	REGION B1.7.2
	    //B1.7.2
	    #"B1.7.2"(ConveyorID := _."B1.7.2",
	              ConveyorSensor:=_."ASiGW-MCC001-bw143-C1: Input"."Sensor B1.7.2",
	              Fault := DB_UDI.ProductionLine.Fault.Stop.Conveyor[_."B1.7.2"],
	              Upstream := DB_UDI.ProductionLine.Upstream.Conveyor[_."B1.7.2"],
	              Downstream := DB_UDI.ProductionLine.DownstreamAccu.Stop.Conveyor[_."B1.7.2"],
	              Interlock := DB_UDI.ProductionLine.Interlock.Stop.Conveyor[_."B1.7.2"],
	              RunForward=>_."ASiGW-MCC001-bw143-C1: Output"."Motor -B1.7.2",
	              WriteAsiDir=>_."ASiGW-MCC001-bw143-C1: Output"."Dir -B1.7.2");
	    
	END_REGION
	
	REGION B1.7.3
	    //B1.7.3
	    #"B1.7.3"(ConveyorID := _."B1.7.3",
	              ConveyorSensor:=_."ASiGW-MCC001-bw143-C1: Input"."Sensor B1.7.3",
	              Fault := DB_UDI.ProductionLine.Fault.Stop.Conveyor[_."B1.7.3"],
	              Upstream := DB_UDI.ProductionLine.Upstream.Conveyor[_."B1.7.3"],
	              Downstream := DB_UDI.ProductionLine.DownstreamAccu.Stop.Conveyor[_."B1.7.3"],
	              Interlock := DB_UDI.ProductionLine.Interlock.Stop.Conveyor[_."B1.7.3"],
	              RunForward=>_."ASiGW-MCC001-bw143-C1: Output"."Motor -B1.7.3",
	              WriteAsiDir=>_."ASiGW-MCC001-bw143-C1: Output"."Dir -B1.7.3");
	    
	END_REGION
	
	REGION B1.8.1
	    //B1.8.1
	    #"B1.8.1"(ConveyorID := _."B1.8.1",
	              ConveyorSensor:=_."ASiGW-MCC001-bw143-C2: Input"."Sensor B1.8.3",
	              Fault := DB_UDI.ProductionLine.Fault.Stop.Conveyor[_."B1.8.1"],
	              Upstream := DB_UDI.ProductionLine.Upstream.Conveyor[_."B1.8.1"],
	              Downstream := DB_UDI.ProductionLine.DownstreamAccu.Stop.Conveyor[_."B1.8.1"],
	              Interlock := DB_UDI.ProductionLine.Interlock.Stop.Conveyor[_."B1.8.1"],
	              RunForward => _."ASiGW-MCC001-bw143-C2: Output"."Motor B1.8.1",
	              WriteAsiDir => _."ASiGW-MCC001-bw143-C2: Output"."Dir B1.8.1");
	    
	END_REGION
	
	REGION B1.8.2
	    //B1.8.2
	    #"B1.8.2"(ConveyorID := _."B1.8.2",
	              ConveyorSensor:=_."ASiGW-MCC001-bw143-C2: Input"."Sensor B1.8.3",
	              Fault := DB_UDI.ProductionLine.Fault.Stop.Conveyor[_."B1.8.2"],
	              Upstream := DB_UDI.ProductionLine.Upstream.Conveyor[_."B1.8.2"],
	              Downstream := DB_UDI.ProductionLine.DownstreamAccu.Stop.Conveyor[_."B1.8.2"],
	              Interlock := DB_UDI.ProductionLine.Interlock.Stop.Conveyor[_."B1.8.2"],
	              RunForward=>_."ASiGW-MCC001-bw143-C2: Output"."Motor B1.8.2",
	              WriteAsiDir=>_."ASiGW-MCC001-bw143-C2: Output"."Dir B1.8.2");
	    
	END_REGION
	
	REGION B1.8.3
	    //B1.8.3
	    #"B1.8.3"(ConveyorID := _."B1.8.3",
	              ConveyorSensor:=_."ASiGW-MCC001-bw143-C2: Input"."Sensor B1.8.3",
	              Fault := DB_UDI.ProductionLine.Fault.Stop.Conveyor[_."B1.8.3"],
	              Upstream := DB_UDI.ProductionLine.Upstream.Conveyor[_."B1.8.3"],
	              Downstream := DB_UDI.ProductionLine.DownstreamAccu.Stop.Conveyor[_."B1.8.3"],
	              Interlock := DB_UDI.ProductionLine.Interlock.Stop.Conveyor[_."B1.8.3"],
	              RunForward=>_."ASiGW-MCC001-bw143-C2: Output"."Motor B1.8.3",
	              WriteAsiDir=>_."ASiGW-MCC001-bw143-C2: Output"."Dir B1.8.3");
	    
	END_REGION
	
	REGION B1.9.1
	    //// B1.9.1 (DP2)
	    #"B1.9.1"(ConveyorID := _."B1.9.1",
	              ConveyorSensor:=_."ASiGW-MCC001-bw143-C2: Input"."Sensor B1.9.1",
	              Fault := DB_UDI.ProductionLine.Fault.Stop.Conveyor[_."B1.9.1"],
	              Upstream := DB_UDI.ProductionLine.Upstream.Conveyor[_."B1.9.1"],
	              Downstream := DB_UDI.ProductionLine.DownstreamAccu.Stop.Conveyor[_."B1.9.1"],
	              Interlock := DB_UDI.ProductionLine.Interlock.Stop.Conveyor[_."B1.9.1"],
	              RunForward=>_."ASiGW-MCC001-bw143-C2: Output"."Motor B1.9.1",
	              WriteAsiDir=>_."ASiGW-MCC001-bw143-C2: Output"."Dir B1.9.1");
	    
	END_REGION
	
	REGION B1.9.2
	    //B1.9.2
	    #"B1.9.2"(ConveyorID := _."B1.9.2",
	              ConveyorSensor:=_."ASiGW-MCC001-bw143-C2: Input"."Sensor B1.9.2",
	              Fault := DB_UDI.ProductionLine.Fault.Stop.Conveyor[_."B1.9.2"],
	              Upstream := DB_UDI.ProductionLine.Upstream.Conveyor[_."B1.9.2"],
	              Downstream := DB_UDI.ProductionLine.DownstreamAccu.Stop.Conveyor[_."B1.9.2"],
	              Interlock := DB_UDI.ProductionLine.Interlock.Stop.Conveyor[_."B1.9.2"],
	              RunForward=>_."ASiGW-MCC001-bw143-C2: Output"."Motor B1.9.2",
	              WriteAsiDir=>_."ASiGW-MCC001-bw143-C2: Output"."Dir B1.9.2");
	    
	END_REGION
	
	REGION B1.10.1 Transfer Unit
	    //// Transfer B1.10.1
	    #"B1.10.1"(TransferID := _."B1.10.1",
	               TransferSensor:=_."ASiGW-MCC001-bw143-C2: Input"."LoadPresence -B1.10.1",
	               Fault := DB_UDI.ProductionLine.Fault.Stop.Conveyor[_."B1.10.1"],
	               Upstream := DB_UDI.ProductionLine.Upstream.Conveyor[_."B1.10.1"],
	               FrontSensor:=_."ASiGW-MCC001-bw143-C2: Input"."FrontSensor -B1.10.1",
	               EndSensor:=_."ASiGW-MCC001-bw143-C2: Input"."EndSensor -B1.10.1",
	               "Left/RightSensor":=_."ASiGW-MCC001-bw143-C2: Input"."LeftSensor -B1.10.1",
	               Downstream := DB_UDI.ProductionLine.DownstreamAccu.Stop.Conveyor[_."B1.10.1"],
	               TransferDirection := DB_ToteTracking.Conveyor[_."B1.10.1"].ToteDir,
	               StartSignal => _."ASiGW-MCC001-bw143-C2: Output"."StartSignal -B1.10.1",
	               Cmd1 => _."ASiGW-MCC001-bw143-C2: Output"."Command1 -B1.10.1",
	               Cmd2 => _."ASiGW-MCC001-bw143-C2: Output"."Command2 -B1.10.1",
	               ErrorReset => _."ASiGW-MCC001-bw143-C2: Output"."ErrorReset -B1.10.1");
	    
	END_REGION
	
	REGION B1.11.1
	    //// B1.11.1 (Go straight TR_B1.11.1)
	    #"B1.11.1"(ConveyorID := _."B1.11.1",
	               ConveyorSensor:=_."ASiGW-MCC001-bw143-C2: Input"."Sensor B1.11.1",
	               Fault := DB_UDI.ProductionLine.Fault.Stop.Conveyor[_."B1.11.1"],
	               Upstream := DB_UDI.ProductionLine.Upstream.Conveyor[_."B1.11.1"],
	               Downstream := DB_UDI.ProductionLine.DownstreamAccu.Stop.Conveyor[_."B1.11.1"],
	               Interlock := DB_UDI.ProductionLine.Interlock.Stop.Conveyor[_."B1.11.1"],
	               RunForward=>_."ASiGW-MCC001-bw143-C2: Output"."Motor B1.11.1",
	               WriteAsiDir=>_."ASiGW-MCC001-bw143-C2: Output"."Dir B1.11.1");
	    
	END_REGION
	
	REGION B1.11.2
	    //B1.11.2
	    #"B1.11.2"(ConveyorID := _."B1.11.2",
	               ConveyorSensor:=_."ASiGW-MCC001-bw143-C2: Input"."Sensor B1.11.4",
	               Fault := DB_UDI.ProductionLine.Fault.Stop.Conveyor[_."B1.11.2"],
	               Upstream := DB_UDI.ProductionLine.Upstream.Conveyor[_."B1.11.2"],
	               Downstream := DB_UDI.ProductionLine.DownstreamAccu.Stop.Conveyor[_."B1.11.2"],
	               Interlock := DB_UDI.ProductionLine.Interlock.Stop.Conveyor[_."B1.11.2"],
	               RunForward=>_."ASiGW-MCC001-bw143-C2: Output"."Motor B1.11.2",
	               WriteAsiDir=>_."ASiGW-MCC001-bw143-C2: Output"."Dir B1.11.2");
	    
	END_REGION
	
	REGION B1.11.3
	    //B1.11.3
	    #"B1.11.3"(ConveyorID := _."B1.11.3",
	               ConveyorSensor:=_."ASiGW-MCC001-bw143-C2: Input"."Sensor B1.11.4",
	               Fault := DB_UDI.ProductionLine.Fault.Stop.Conveyor[_."B1.11.3"],
	               Upstream := DB_UDI.ProductionLine.Upstream.Conveyor[_."B1.11.3"],
	               Downstream := DB_UDI.ProductionLine.DownstreamAccu.Stop.Conveyor[_."B1.11.3"],
	               Interlock := DB_UDI.ProductionLine.Interlock.Stop.Conveyor[_."B1.11.3"],
	               RunForward=>_."ASiGW-MCC001-bw143-C2: Output"."Motor B1.11.3",
	               WriteAsiDir=>_."ASiGW-MCC001-bw143-C2: Output"."Dir B1.11.3");
	    
	END_REGION
	
	REGION B1.11.4
	    //B1.11.4
	    #"B1.11.4"(ConveyorID := _."B1.11.4",
	               ConveyorSensor:=_."ASiGW-MCC001-bw143-C2: Input"."Sensor B1.11.4",
	               Fault := DB_UDI.ProductionLine.Fault.Stop.Conveyor[_."B1.11.4"],
	               Upstream := DB_UDI.ProductionLine.Upstream.Conveyor[_."B1.11.4"],
	               Downstream := DB_UDI.ProductionLine.DownstreamAccu.Stop.Conveyor[_."B1.11.4"],
	               Interlock := DB_UDI.ProductionLine.Interlock.Stop.Conveyor[_."B1.11.4"],
	               RunForward => _."ASiGW-MCC001-bw143-C2: Output"."Motor B1.11.4",
	               WriteAsiDir => _."ASiGW-MCC001-bw143-C2: Output"."Dir B1.11.4");
	    
	END_REGION
	
	REGION B1.12.1
	    //B1.12.1
	    #"B1.12.1"(ConveyorID := _."B1.12.1",
	               ConveyorSensor:=_."ASiGW-MCC001-bw143-C2: Input"."Sensor B1.12.1",
	               Fault := DB_UDI.ProductionLine.Fault.Stop.Conveyor[_."B1.12.1"],
	               Upstream := DB_UDI.ProductionLine.Upstream.Conveyor[_."B1.12.1"],
	               Downstream := DB_UDI.ProductionLine.DownstreamAccu.Stop.Conveyor[_."B1.12.1"],
	               Interlock := DB_UDI.ProductionLine.Interlock.Stop.Conveyor[_."B1.12.1"],
	               RunForward=>_."ASiGW-MCC001-bw143-C2: Output"."Motor B1.12.1",
	               WriteAsiDir=>_."ASiGW-MCC001-bw143-C2: Output"."Dir B1.12.1");
	    
	END_REGION
	
	REGION B1.12.2
	    //B1.12.2
	    #"B1.12.2"(ConveyorID := _."B1.12.2",
	               ConveyorSensor:=_."ASiGW-MCC001-bw143-C2: Input"."Sensor B1.12.2",
	               Fault := DB_UDI.ProductionLine.Fault.Stop.Conveyor[_."B1.12.2"],
	               Upstream := DB_UDI.ProductionLine.Upstream.Conveyor[_."B1.12.2"],
	               Downstream := DB_UDI.ProductionLine.DownstreamAccu.Stop.Conveyor[_."B1.12.2"],
	               Interlock := DB_UDI.ProductionLine.Interlock.Stop.Conveyor[_."B1.12.2"],
	               RunForward=>_."ASiGW-MCC001-bw143-C2: Output"."Motor B1.12.2",
	               WriteAsiDir=>_."ASiGW-MCC001-bw143-C2: Output"."Dir B1.12.2");
	    
	END_REGION
	
	REGION B1.13.1 Transfer Unit
	    //// Transfer B1.13.1
	    #"B1.13.1"(TransferID := _."B1.13.1",
	               TransferSensor:=_."ASiGW-MCC001-bw143-C2: Input"."LoadPresence -B1.13.1",
	               Fault := DB_UDI.ProductionLine.Fault.Stop.Conveyor[_."B1.13.1"],
	               Upstream := DB_UDI.ProductionLine.Upstream.Conveyor[_."B1.13.1"],
	               FrontSensor:=_."ASiGW-MCC001-bw143-C2: Input"."FrontSensor -B1.13.1",
	               EndSensor:=_."ASiGW-MCC001-bw143-C2: Input"."EndSensor -B1.13.1",
	               "Left/RightSensor":=_."ASiGW-MCC001-bw143-C2: Input"."LeftSensor -B1.13.1",
	               Downstream := DB_UDI.ProductionLine.DownstreamAccu.Stop.Conveyor[_."B1.13.1"],
	               TransferDirection := DB_ToteTracking.Conveyor[_."B1.13.1"].ToteDir,
	               StartSignal => _."ASiGW-MCC001-bw143-C2: Output"."StartSignal - B1.13.1",
	               Cmd1 => _."ASiGW-MCC001-bw143-C2: Output"."Command1 -B1.13.1",
	               Cmd2 => _."ASiGW-MCC001-bw143-C2: Output"."Command2 -B1.13.1",
	               ErrorReset => _."ASiGW-MCC001-bw143-C2: Output"."ErrorReset -B1.13.1");
	    
	END_REGION
	
	REGION B1.14.1 Transfer Unit
	    //// Transfer B1.14.1
	    #"B1.14.1"(TransferID := _."B1.14.1",
	               TransferSensor:=_."ASiGW-MCC001-bw143-C2: Input"."LoadPresence -B1.14.1",
	               Fault := DB_UDI.ProductionLine.Fault.Stop.Conveyor[_."B1.14.1"],
	               Upstream := DB_UDI.ProductionLine.Upstream.Conveyor[_."B1.14.1"],
	               FrontSensor:=_."ASiGW-MCC001-bw143-C2: Input"."FrontSensor -B1.14.1",
	               EndSensor:=_."ASiGW-MCC001-bw143-C2: Input"."EndSensor -B1.14.1",
	               "Left/RightSensor":=_."ASiGW-MCC001-bw143-C2: Input"."LeftSensor -B1.14.1",
	               Downstream := DB_UDI.ProductionLine.DownstreamAccu.Stop.Conveyor[_."B1.14.1"],
	               TransferDirection := DB_ToteTracking.Conveyor[_."B1.14.1"].ToteDir,
	               StartSignal => _."ASiGW-MCC001-bw143-C2: Output"."StartSignal -B1.14.1",
	               Cmd1 => _."ASiGW-MCC001-bw143-C2: Output"."Command1 -B1.14.1",
	               Cmd2 => _."ASiGW-MCC001-bw143-C2: Output"."Command2 -B1.14.1",
	               ErrorReset => _."ASiGW-MCC001-bw143-C2: Output"."ErrorReset -B1.14.1");
	    
	END_REGION
	
	REGION B1.15.1
	    //// B1.15.1 (Go straight TR_B1.17.1)
	    #"B1.15.1"(ConveyorID := _."B1.15.1",
	               ConveyorSensor:=_."ASiGW-MCC001-bw143-C2: Input"."Sensor B1.15.1",
	               Fault := DB_UDI.ProductionLine.Fault.Stop.Conveyor[_."B1.15.1"],
	               Upstream := DB_UDI.ProductionLine.Upstream.Conveyor[_."B1.15.1"],
	               Downstream := DB_UDI.ProductionLine.DownstreamAccu.Stop.Conveyor[_."B1.15.1"],
	               Interlock := DB_UDI.ProductionLine.Interlock.Stop.Conveyor[_."B1.15.1"],
	               RunForward=>_."ASiGW-MCC001-bw143-C2: Output"."Motor B1.15.1",
	               WriteAsiDir=>_."ASiGW-MCC001-bw143-C2: Output"."Dir B1.15.1");
	    
	END_REGION
	
	REGION B1.15.2
	    //B1.15.2
	    #"B1.15.2"(ConveyorID := _."B1.15.2",
	               ConveyorSensor:=_."ASiGW-MCC001-bw143-C2: Input"."Sensor B1.15.2",
	               Fault := DB_UDI.ProductionLine.Fault.Stop.Conveyor[_."B1.15.2"],
	               Upstream := DB_UDI.ProductionLine.Upstream.Conveyor[_."B1.15.2"],
	               Downstream := DB_UDI.ProductionLine.DownstreamAccu.Stop.Conveyor[_."B1.15.2"],
	               Interlock := DB_UDI.ProductionLine.Interlock.Stop.Conveyor[_."B1.15.2"],
	               RunForward=>_."ASiGW-MCC001-bw143-C2: Output"."Motor B1.15.2",
	               WriteAsiDir=>_."ASiGW-MCC001-bw143-C2: Output"."Dir B1.15.2");
	    
	END_REGION
	
	REGION B1.16.1
	    //B1.16.1
	    #"B1.16.1"(ConveyorID := _."B1.16.1",
	               ConveyorSensor:=_."ASiGW-MCC001-bw143-C2: Input"."Sensor B1.16.8",
	               Fault := DB_UDI.ProductionLine.Fault.Stop.Conveyor[_."B1.16.1"],
	               Upstream := DB_UDI.ProductionLine.Upstream.Conveyor[_."B1.16.1"],
	               Downstream := DB_UDI.ProductionLine.DownstreamAccu.Stop.Conveyor[_."B1.16.1"],
	               Interlock := DB_UDI.ProductionLine.Interlock.Stop.Conveyor[_."B1.16.1"],
	               RunForward => _."ASiGW-MCC001-bw143-C2: Output"."Motor B1.16.1",
	               WriteAsiDir => _."ASiGW-MCC001-bw143-C2: Output"."Dir B1.16.1");
	    
	END_REGION
	
	REGION B1.16.2
	    //B1.16.2
	    #"B1.16.2"(ConveyorID := _."B1.16.2",
	               ConveyorSensor:=_."ASiGW-MCC001-bw143-C2: Input"."Sensor B1.16.8",
	               Fault := DB_UDI.ProductionLine.Fault.Stop.Conveyor[_."B1.16.2"],
	               Upstream := DB_UDI.ProductionLine.Upstream.Conveyor[_."B1.16.2"],
	               Downstream := DB_UDI.ProductionLine.DownstreamAccu.Stop.Conveyor[_."B1.16.2"],
	               Interlock := DB_UDI.ProductionLine.Interlock.Stop.Conveyor[_."B1.16.2"],
	               RunForward=>_."ASiGW-MCC001-bw143-C2: Output"."Motor B1.16.2",
	               WriteAsiDir=>_."ASiGW-MCC001-bw143-C2: Output"."Dir B1.16.2");
	    
	END_REGION
	
	REGION B1.16.3
	    //B1.16.3
	    #"B1.16.3"(ConveyorID := _."B1.16.3",
	               ConveyorSensor:=_."ASiGW-MCC001-bw143-C2: Input"."Sensor B1.16.8",
	               Fault := DB_UDI.ProductionLine.Fault.Stop.Conveyor[_."B1.16.3"],
	               Upstream := DB_UDI.ProductionLine.Upstream.Conveyor[_."B1.16.3"],
	               Downstream := DB_UDI.ProductionLine.DownstreamAccu.Stop.Conveyor[_."B1.16.3"],
	               Interlock := DB_UDI.ProductionLine.Interlock.Stop.Conveyor[_."B1.16.3"],
	               RunForward=>_."ASiGW-MCC001-bw143-C2: Output"."Motor B1.16.3",
	               WriteAsiDir=>_."ASiGW-MCC001-bw143-C2: Output"."Dir B1.16.3");
	    
	END_REGION
	
	REGION B1.16.4
	    //B1.16.4
	    #"B1.16.4"(ConveyorID := _."B1.16.4",
	               ConveyorSensor:=_."ASiGW-MCC001-bw143-C2: Input"."Sensor B1.16.8",
	               Fault := DB_UDI.ProductionLine.Fault.Stop.Conveyor[_."B1.16.4"],
	               Upstream := DB_UDI.ProductionLine.Upstream.Conveyor[_."B1.16.4"],
	               Downstream := DB_UDI.ProductionLine.DownstreamAccu.Stop.Conveyor[_."B1.16.4"],
	               Interlock := DB_UDI.ProductionLine.Interlock.Stop.Conveyor[_."B1.16.4"],
	               RunForward=>_."ASiGW-MCC001-bw143-C2: Output"."Motor B1.16.4",
	               WriteAsiDir=>_."ASiGW-MCC001-bw143-C2: Output"."Dir B1.16.4");
	    
	END_REGION
	
	REGION B1.16.5
	    //B1.16.5
	    #"B1.16.5"(ConveyorID := _."B1.16.5",
	               ConveyorSensor:=_."ASiGW-MCC001-bw143-C2: Input"."Sensor B1.16.8",
	               Fault := DB_UDI.ProductionLine.Fault.Stop.Conveyor[_."B1.16.5"],
	               Upstream := DB_UDI.ProductionLine.Upstream.Conveyor[_."B1.16.5"],
	               Downstream := DB_UDI.ProductionLine.DownstreamAccu.Stop.Conveyor[_."B1.16.5"],
	               Interlock := DB_UDI.ProductionLine.Interlock.Stop.Conveyor[_."B1.16.5"],
	               RunForward=>_."ASiGW-MCC001-bw143-C2: Output"."Motor B1.16.5",
	               WriteAsiDir=>_."ASiGW-MCC001-bw143-C2: Output"."Dir B1.16.5");
	    
	END_REGION
	
	REGION B1.16.6
	    //B1.16.6
	    #"B1.16.6"(ConveyorID := _."B1.16.6",
	               ConveyorSensor:=_."ASiGW-MCC001-bw143-C2: Input"."Sensor B1.16.8",
	               Fault := DB_UDI.ProductionLine.Fault.Stop.Conveyor[_."B1.16.6"],
	               Upstream := DB_UDI.ProductionLine.Upstream.Conveyor[_."B1.16.6"],
	               Downstream := DB_UDI.ProductionLine.DownstreamAccu.Stop.Conveyor[_."B1.16.6"],
	               Interlock := DB_UDI.ProductionLine.Interlock.Stop.Conveyor[_."B1.16.6"],
	               RunForward=>_."ASiGW-MCC001-bw143-C2: Output"."Motor B1.16.6",
	               WriteAsiDir=>_."ASiGW-MCC001-bw143-C2: Output"."Dir B1.16.6");
	    
	END_REGION
	
	REGION B1.16.7
	    //B1.16.7
	    #"B1.16.7"(ConveyorID := _."B1.16.7",
	               ConveyorSensor:=_."ASiGW-MCC001-bw143-C2: Input"."Sensor B1.16.8",
	               Fault := DB_UDI.ProductionLine.Fault.Stop.Conveyor[_."B1.16.7"],
	               Upstream := DB_UDI.ProductionLine.Upstream.Conveyor[_."B1.16.7"],
	               Downstream := DB_UDI.ProductionLine.DownstreamAccu.Stop.Conveyor[_."B1.16.7"],
	               Interlock := DB_UDI.ProductionLine.Interlock.Stop.Conveyor[_."B1.16.7"],
	               RunForward => _."ASiGW-MCC001-bw143-C2: Output"."Motor B1.16.7",
	               WriteAsiDir => _."ASiGW-MCC001-bw143-C2: Output"."Dir B1.16.7");
	    
	END_REGION
	
	REGION B1.16.8
	    //B1.16.8
	    #"B1.16.8"(ConveyorID := _."B1.16.8",
	               ConveyorSensor:=_."ASiGW-MCC001-bw143-C2: Input"."Sensor B1.16.8",
	               Fault := DB_UDI.ProductionLine.Fault.Stop.Conveyor[_."B1.16.8"],
	               Upstream := DB_UDI.ProductionLine.Upstream.Conveyor[_."B1.16.8"],
	               Downstream := DB_UDI.ProductionLine.DownstreamAccu.Stop.Conveyor[_."B1.16.8"],
	               Interlock := DB_UDI.ProductionLine.Interlock.Stop.Conveyor[_."B1.16.8"],
	               RunForward=>_."ASiGW-MCC001-bw143-C2: Output"."Motor B1.16.8",
	               WriteAsiDir=>_."ASiGW-MCC001-bw143-C2: Output"."Dir B1.16.8");
	    
	END_REGION
	
	REGION B1.17.1
	    //// B1.17.1 (DP3)
	    #"B1.17.1"(ConveyorID := _."B1.17.1",
	               ConveyorSensor:=_."ASiGW-MCC001-bw143-C2: Input"."Sensor B1.17.1",
	               Fault := DB_UDI.ProductionLine.Fault.Stop.Conveyor[_."B1.17.1"],
	               Upstream := DB_UDI.ProductionLine.Upstream.Conveyor[_."B1.17.1"],
	               Downstream := DB_UDI.ProductionLine.DownstreamAccu.Stop.Conveyor[_."B1.17.1"],
	               Interlock := DB_UDI.ProductionLine.Interlock.Stop.Conveyor[_."B1.17.1"],
	               RunForward => _."ASiGW-MCC001-bw143-C2: Output"."Motor B1.17.1",
	               WriteAsiDir => _."ASiGW-MCC001-bw143-C2: Output"."Dir B1.17.1");
	    
	END_REGION
	
	REGION B1.17.2
	    //B1.17.2
	    #"B1.17.2"(ConveyorID := _."B1.17.2",
	               ConveyorSensor:=_."ASiGW-MCC001-bw143-C2: Input"."Sensor B1.17.2",
	               Fault := DB_UDI.ProductionLine.Fault.Stop.Conveyor[_."B1.17.2"],
	               Upstream := DB_UDI.ProductionLine.Upstream.Conveyor[_."B1.17.2"],
	               Downstream := DB_UDI.ProductionLine.DownstreamAccu.Stop.Conveyor[_."B1.17.2"],
	               Interlock := DB_UDI.ProductionLine.Interlock.Stop.Conveyor[_."B1.17.2"],
	               RunForward => _."ASiGW-MCC001-bw143-C2: Output"."Motor B1.17.2",
	               WriteAsiDir => _."ASiGW-MCC001-bw143-C2: Output"."Dir B1.17.2");
	    
	END_REGION
	
	REGION B1.17.3
	    //B1.17.3
	    #"B1.17.3"(ConveyorID := _."B1.17.3",
	               ConveyorSensor:=_."ASiGW-MCC001-bw143-C2: Input"."Sensor B1.17.3",
	               Fault := DB_UDI.ProductionLine.Fault.Stop.Conveyor[_."B1.17.3"],
	               Upstream := DB_UDI.ProductionLine.Upstream.Conveyor[_."B1.17.3"],
	               Downstream := DB_UDI.ProductionLine.DownstreamAccu.Stop.Conveyor[_."B1.17.3"],
	               Interlock := DB_UDI.ProductionLine.Interlock.Stop.Conveyor[_."B1.17.3"],
	               RunForward => _."ASiGW-MCC001-bw143-C2: Output"."Motor B1.17.3",
	               WriteAsiDir => _."ASiGW-MCC001-bw143-C2: Output"."Dir B1.17.3");
	    
	END_REGION
	
	REGION B1.17.4
	    //B1.17.4
	    #"B1.17.4"(ConveyorID := _."B1.17.4",
	               ConveyorSensor:=_."ASiGW-MCC001-bw143-C2: Input"."Sensor B1.17.4",
	               Fault := DB_UDI.ProductionLine.Fault.Stop.Conveyor[_."B1.17.4"],
	               Upstream := DB_UDI.ProductionLine.Upstream.Conveyor[_."B1.17.4"],
	               Downstream := DB_UDI.ProductionLine.DownstreamAccu.Stop.Conveyor[_."B1.17.4"],
	               Interlock := DB_UDI.ProductionLine.Interlock.Stop.Conveyor[_."B1.17.4"],
	               RunForward => _."ASiGW-MCC001-bw143-C2: Output"."Motor B1.17.4",
	               WriteAsiDir => _."ASiGW-MCC001-bw143-C2: Output"."Dir B1.17.4");
	    
	END_REGION
	
	REGION B1.18.1 Transfer Unit
	    //// Transfer B1.18.1
	    #"B1.18.1"(TransferID := _."B1.18.1",
	               TransferSensor:=_."ASiGW-MCC001-bw143-C2: Input"."LoadPresence -B1.18.1",
	               Fault := DB_UDI.ProductionLine.Fault.Stop.Conveyor[_."B1.18.1"],
	               Upstream := DB_UDI.ProductionLine.Upstream.Conveyor[_."B1.18.1"],
	               FrontSensor:=_."ASiGW-MCC001-bw143-C2: Input"."FrontSensor -B1.18.1",
	               EndSensor:=_."ASiGW-MCC001-bw143-C2: Input"."EndSensor -B1.18.1",
	               "Left/RightSensor":=_."ASiGW-MCC001-bw143-C2: Input"."LeftSensor -B1.18.1",
	               Downstream := DB_UDI.ProductionLine.DownstreamAccu.Stop.Conveyor[_."B1.18.1"],
	               TransferDirection := DB_ToteTracking.Conveyor[_."B1.18.1"].ToteDir,
	               StartSignal => _."ASiGW-MCC001-bw143-C2: Output"."StartSignal -B1.18.1",
	               Cmd1 => _."ASiGW-MCC001-bw143-C2: Output"."Command1 -B1.18.1",
	               Cmd2 => _."ASiGW-MCC001-bw143-C2: Output"."Command2 -B1.18.1",
	               ErrorReset => _."ASiGW-MCC001-bw143-C2: Output"."ErrorReset -B1.18.1");
	    
	END_REGION
	
	REGION B1.19.1
	    //B1.19.1
	    #"B1.19.1"(ConveyorID := _."B1.19.1",
	               ConveyorSensor:=_."ASiGW-MCC001-bw143-C2: Input"."Sensor B1.19.1",
	               Fault := DB_UDI.ProductionLine.Fault.Stop.Conveyor[_."B1.19.1"],
	               Upstream := DB_UDI.ProductionLine.Upstream.Conveyor[_."B1.19.1"],
	               Downstream := DB_UDI.ProductionLine.DownstreamAccu.Stop.Conveyor[_."B1.19.1"],
	               Interlock := DB_UDI.ProductionLine.Interlock.Stop.Conveyor[_."B1.19.1"],
	               RunForward => _."ASiGW-MCC001-bw143-C2: Output"."Motor B1.19.1",
	               WriteAsiDir => _."ASiGW-MCC001-bw143-C2: Output"."Dir B1.19.1");
	    
	END_REGION
	
	REGION B1.20.1
	    //B1.20.1
	    #"B1.20.1"(ConveyorID := _."B1.20.1",
	               ConveyorSensor:=_."ASiGW-MCC001-bw143-C2: Input"."Sensor B1.20.1",
	               Fault := DB_UDI.ProductionLine.Fault.Stop.Conveyor[_."B1.20.1"],
	               Upstream := DB_UDI.ProductionLine.Upstream.Conveyor[_."B1.20.1"],
	               Downstream := DB_UDI.ProductionLine.DownstreamAccu.Stop.Conveyor[_."B1.20.1"],
	               Interlock := DB_UDI.ProductionLine.Interlock.Stop.Conveyor[_."B1.20.1"],
	               RunForward => _."ASiGW-MCC001-bw143-C2: Output"."Motor B1.20.1",
	               WriteAsiDir => _."ASiGW-MCC001-bw143-C2: Output"."Dir B1.20.1");
	    
	END_REGION
	
	REGION B1.20.2
	    //B1.20.2
	    #"B1.20.2"(ConveyorID := _."B1.20.2",
	               ConveyorSensor:=_."ASiGW-MCC001-bw143-C2: Input"."Sensor B1.20.2",
	               Fault := DB_UDI.ProductionLine.Fault.Stop.Conveyor[_."B1.20.2"],
	               Upstream := DB_UDI.ProductionLine.Upstream.Conveyor[_."B1.20.2"],
	               Downstream := DB_UDI.ProductionLine.DownstreamAccu.Stop.Conveyor[_."B1.20.2"],
	               Interlock := DB_UDI.ProductionLine.Interlock.Stop.Conveyor[_."B1.20.2"],
	               RunForward => _."ASiGW-MCC001-bw143-C2: Output"."Motor B1.20.2",
	               WriteAsiDir => _."ASiGW-MCC001-bw143-C2: Output"."Dir B1.20.2");
	    
	END_REGION
	
	REGION B1.21.1
	    //B1.21.1
	    #"B1.21.1"(ConveyorID := _."B1.21.1",
	               ConveyorSensor:=_."ASiGW-MCC001-bw143-C2: Input"."Sensor B1.21.1",
	               Fault := DB_UDI.ProductionLine.Fault.Stop.Conveyor[_."B1.21.1"],
	               Upstream := DB_UDI.ProductionLine.Upstream.Conveyor[_."B1.21.1"],
	               Downstream := DB_UDI.ProductionLine.DownstreamAccu.Stop.Conveyor[_."B1.21.1"],
	               Interlock := DB_UDI.ProductionLine.Interlock.Stop.Conveyor[_."B1.21.1"],
	               RunForward => _."ASiGW-MCC001-bw143-C2: Output"."Motor B1.21.1",
	               WriteAsiDir => _."ASiGW-MCC001-bw143-C2: Output"."Dir B1.21.1");
	    
	END_REGION
	
	REGION B1.21.2
	    //B1.21.2
	    #"B1.21.2"(ConveyorID := _."B1.21.2",
	               ConveyorSensor:=_."ASiGW-MCC001-bw143-C2: Input"."Sensor B1.21.2",
	               Fault := DB_UDI.ProductionLine.Fault.Stop.Conveyor[_."B1.21.2"],
	               Upstream := DB_UDI.ProductionLine.Upstream.Conveyor[_."B1.21.2"],
	               Downstream := DB_UDI.ProductionLine.DownstreamAccu.Stop.Conveyor[_."B1.21.2"],
	               Interlock := DB_UDI.ProductionLine.Interlock.Stop.Conveyor[_."B1.21.2"],
	               RunForward => _."ASiGW-MCC001-bw143-C2: Output"."Motor B1.21.2",
	               WriteAsiDir => _."ASiGW-MCC001-bw143-C2: Output"."Dir B1.21.2");
	    
	END_REGION
	
	REGION B1.21.3
	    //B1.21.3
	    #"B1.21.3"(ConveyorID := _."B1.21.3",
	               ConveyorSensor:=_."ASiGW-MCC001-bw143-C2: Input"."Sensor B1.23.1",
	               Fault := DB_UDI.ProductionLine.Fault.Stop.Conveyor[_."B1.21.3"],
	               Upstream := DB_UDI.ProductionLine.Upstream.Conveyor[_."B1.21.3"],
	               Downstream := DB_UDI.ProductionLine.DownstreamAccu.Stop.Conveyor[_."B1.21.3"],
	               Interlock := DB_UDI.ProductionLine.Interlock.Stop.Conveyor[_."B1.21.3"],
	               RunForward => _."ASiGW-MCC001-bw143-C2: Output"."Motor B1.21.3",
	               WriteAsiDir => _."ASiGW-MCC001-bw143-C2: Output"."Dir B1.21.3");
	    
	END_REGION
	
	REGION B1.22.1
	    //B1.22.1
	    #"B1.22.1"(ConveyorID := _."B1.22.1",
	               ConveyorSensor:=_."ASiGW-MCC001-bw143-C2: Input"."Sensor B1.23.1",
	               Fault := DB_UDI.ProductionLine.Fault.Stop.Conveyor[_."B1.22.1"],
	               Upstream := DB_UDI.ProductionLine.Upstream.Conveyor[_."B1.22.1"],
	               Downstream := DB_UDI.ProductionLine.DownstreamAccu.Stop.Conveyor[_."B1.22.1"],
	               Interlock := DB_UDI.ProductionLine.Interlock.Stop.Conveyor[_."B1.22.1"],
	               RunForward => _."ASiGW-MCC001-bw143-C2: Output"."Motor - B1.22.1",
	               WriteAsiDir => _."ASiGW-MCC001-bw143-C2: Output"."2-30A Dir",
	               WriteAsiSpeed => _."ASiGW-MCC001-bw143-C2: Output"."2-30A Speed");
	    
	END_REGION
	
	REGION B1.23.1
	    ////B1.23.1 Arm for Merger1
	    #"B1.23.1"(ConveyorID := _."B1.23.1",
	               ConveyorSensor:=_."ASiGW-MCC001-bw143-C2: Input"."Sensor B1.23.1",
	               Fault := DB_UDI.ProductionLine.Fault.Stop.Conveyor[_."B1.23.1"],
	               Upstream := DB_UDI.ProductionLine.Upstream.Conveyor[_."B1.23.1"],
	               Downstream := DB_UDI.ProductionLine.DownstreamAccu.Stop.Conveyor[_."B1.23.1"],
	               Interlock := DB_UDI.ProductionLine.Interlock.Stop.Conveyor[_."B1.23.1"],
	               RunForward => _."ASiGW-MCC001-bw143-C2: Output"."Motor B1.23.1",
	               WriteAsiDir => _."ASiGW-MCC001-bw143-C2: Output"."Dir B1.23.1");
	    
	END_REGION
	
	REGION C1.3.1 Transfer Unit
	    ////Transfer C1.3.1
	    #"C1.3.1"(TransferID := _."C1.3.1",
	              TransferSensor:=_."ASiGW-MCC001-bw143-C2: Input"."LoadPresence -C1.3.1",
	              Fault := DB_UDI.ProductionLine.Fault.Stop.Conveyor[_."C1.3.1"],
	              Upstream := DB_UDI.ProductionLine.Upstream.Conveyor[_."C1.3.1"],
	              FrontSensor:=_."ASiGW-MCC001-bw143-C2: Input"."FrontSensor -C1.3.1",
	              EndSensor:=_."ASiGW-MCC001-bw143-C2: Input"."EndSensor -C1.3.1",
	              "Left/RightSensor":=_."ASiGW-MCC001-bw143-C2: Input"."LeftSensor -C1.3.1",
	              Downstream := DB_UDI.ProductionLine.DownstreamAccu.Stop.Conveyor[_."C1.3.1"],
	              TransferDirection := DB_ToteTracking.Conveyor[_."C1.3.1"].ToteDir,
	              StartSignal => _."ASiGW-MCC001-bw143-C2: Output"."StartSignal -C1.3.1",
	              Cmd1 => _."ASiGW-MCC001-bw143-C2: Output"."Command1 -C1.3.1",
	              Cmd2 => _."ASiGW-MCC001-bw143-C2: Output"."Command2 -C1.3.1",
	              ErrorReset => _."ASiGW-MCC001-bw143-C2: Output"."ErrorReset -C1.3.1");
	    
	END_REGION
	
	REGION C1.2.2
	    //// C1.2.2  (Go Right TR_C1.1.3)
	    #"C1.2.2"(ConveyorID := _."C1.2.2",
	              ConveyorSensor:=_."ASiGW-MCC001-bw143-C2: Input"."Sensor C1.2.2",
	              Fault := DB_UDI.ProductionLine.Fault.Stop.Conveyor[_."C1.2.2"],
	              Upstream := DB_UDI.ProductionLine.Upstream.Conveyor[_."C1.2.2"],
	              Downstream := DB_UDI.ProductionLine.DownstreamAccu.Stop.Conveyor[_."C1.2.2"],
	              Interlock := DB_UDI.ProductionLine.Interlock.Stop.Conveyor[_."C1.2.2"],
	              RunForward=>_."ASiGW-MCC001-bw143-C2: Output"."Motor C1.2.2",
	              WriteAsiDir=>_."ASiGW-MCC001-bw143-C2: Output"."Dir C1.2.2");
	    
	END_REGION
	
	REGION C1.2.1
	    //C1.2.1
	    #"C1.2.1"(ConveyorID := _."C1.2.1",
	              ConveyorSensor:=_."ASiGW-MCC001-bw143-C2: Input"."Sensor C1.2.1",
	              Fault := DB_UDI.ProductionLine.Fault.Stop.Conveyor[_."C1.2.1"],
	              Upstream := DB_UDI.ProductionLine.Upstream.Conveyor[_."C1.2.1"],
	              Downstream := DB_UDI.ProductionLine.DownstreamAccu.Stop.Conveyor[_."C1.2.1"],
	              Interlock := DB_UDI.ProductionLine.Interlock.Stop.Conveyor[_."C1.2.1"],
	              RunForward=>_."ASiGW-MCC001-bw143-C2: Output"."Motor C1.2.1",
	              WriteAsiDir=>_."ASiGW-MCC001-bw143-C2: Output"."Dir C1.2.1");
	    
	END_REGION
	
	REGION C1.4.1
	    //// C1.4.1  (Go Left TR_C1.1.3)
	    #"C1.4.1"(ConveyorID := _."C1.4.1",
	              ConveyorSensor:=_."ASiGW-MCC001-bw143-C2: Input"."Sensor C1.4.1",
	              Fault := DB_UDI.ProductionLine.Fault.Stop.Conveyor[_."C1.4.1"],
	              Upstream := DB_UDI.ProductionLine.Upstream.Conveyor[_."C1.4.1"],
	              Downstream := DB_UDI.ProductionLine.DownstreamAccu.Stop.Conveyor[_."C1.4.1"],
	              Interlock := DB_UDI.ProductionLine.Interlock.Stop.Conveyor[_."C1.4.1"],
	              RunForward=>_."ASiGW-MCC001-bw143-C2: Output"."Motor C1.4.1",
	              WriteAsiDir=>_."ASiGW-MCC001-bw143-C2: Output"."Dir C1.4.1");
	    
	END_REGION
	
	REGION C1.4.2
	    //C1.4.2
	    #"C1.4.2"(ConveyorID := _."C1.4.2",
	              ConveyorSensor:=_."ASiGW-MCC001-bw143-C2: Input"."Sensor C1.4.2",
	              Fault := DB_UDI.ProductionLine.Fault.Stop.Conveyor[_."C1.4.2"],
	              Upstream := DB_UDI.ProductionLine.Upstream.Conveyor[_."C1.4.2"],
	              Downstream := DB_UDI.ProductionLine.DownstreamAccu.Stop.Conveyor[_."C1.4.2"],
	              Interlock := DB_UDI.ProductionLine.Interlock.Stop.Conveyor[_."C1.4.2"],
	              RunForward=>_."ASiGW-MCC001-bw143-C2: Output"."Motor C1.4.2",
	              WriteAsiDir=>_."ASiGW-MCC001-bw143-C2: Output"."Dir C1.4.2");
	    
	END_REGION
	
	REGION D1.1.1
	    ////  D1.1.1 (Go Right DP4)
	    #"D1.1.1"(ConveyorID := _."D1.1.1",
	              ConveyorSensor:=_."ASiGW-MCC001-bw200-C1: Input"."Sensor D1.2.1",
	              Fault := DB_UDI.ProductionLine.Fault.Stop.Conveyor[_."D1.1.1"],
	              Upstream := DB_UDI.ProductionLine.Upstream.Conveyor[_."D1.1.1"],
	              Downstream := DB_UDI.ProductionLine.DownstreamAccu.Stop.Conveyor[_."D1.1.1"],
	              Interlock := DB_UDI.ProductionLine.Interlock.Stop.Conveyor[_."D1.1.1"],
	              RunForward=>_."ASiGW-MCC001-bw200-C1: Output"."Motor D1.1.1",
	              WriteAsiDir=>_."ASiGW-MCC001-bw200-C1: Output"."Dir D1.1.1");
	    
	END_REGION
	
	REGION D1.2.1
	    //D1.2.1
	    #"D1.2.1"(ConveyorID := _."D1.2.1",
	              ConveyorSensor:=_."ASiGW-MCC001-bw200-C1: Input"."Sensor D1.2.1",
	              Fault := DB_UDI.ProductionLine.Fault.Stop.Conveyor[_."D1.2.1"],
	              Upstream := DB_UDI.ProductionLine.Upstream.Conveyor[_."D1.2.1"],
	              Downstream := DB_UDI.ProductionLine.DownstreamAccu.Stop.Conveyor[_."D1.2.1"],
	              Interlock := DB_UDI.ProductionLine.Interlock.Stop.Conveyor[_."D1.2.1"],
	              RunForward=>_."ASiGW-MCC001-bw200-C1: Output"."Motor - D1.2.1",
	              WriteAsiDir=>_."ASiGW-MCC001-bw200-C1: Output"."1-2A Dir",
	              WriteAsiSpeed=>_."ASiGW-MCC001-bw200-C1: Output"."1-2A Speed");
	    
	END_REGION
	
	REGION D1.3.1
	    //D1.3.1
	    #"D1.3.1"(ConveyorID := _."D1.3.1",
	              ConveyorSensor:=_."ASiGW-MCC001-bw200-C1: Input"."Sensor D1.3.1",
	              Fault := DB_UDI.ProductionLine.Fault.Stop.Conveyor[_."D1.3.1"],
	              Upstream := DB_UDI.ProductionLine.Upstream.Conveyor[_."D1.3.1"],
	              Downstream := DB_UDI.ProductionLine.DownstreamAccu.Stop.Conveyor[_."D1.3.1"],
	              Interlock := DB_UDI.ProductionLine.Interlock.Stop.Conveyor[_."D1.3.1"],
	              RunForward=>_."ASiGW-MCC001-bw200-C1: Output"."Motor - D1.3.1",
	              WriteAsiDir=>_."ASiGW-MCC001-bw200-C1: Output"."1-2A Dir",
	              WriteAsiSpeed=>_."ASiGW-MCC001-bw200-C1: Output"."1-2A Speed");
	    
	END_REGION
	
	REGION D1.4.1
	    //D1.4.1
	    #"D1.4.1"(ConveyorID := _."D1.4.1",
	              ConveyorSensor:=_."ASiGW-MCC001-bw200-C1: Input"."Sensor D1.4.1",
	              Fault := DB_UDI.ProductionLine.Fault.Stop.Conveyor[_."D1.4.1"],
	              Upstream := DB_UDI.ProductionLine.Upstream.Conveyor[_."D1.4.1"],
	              Downstream := DB_UDI.ProductionLine.DownstreamAccu.Stop.Conveyor[_."D1.4.1"],
	              Interlock := DB_UDI.ProductionLine.Interlock.Stop.Conveyor[_."D1.4.1"],
	              RunForward=>_."ASiGW-MCC001-bw200-C1: Output"."Motor D1.4.1",
	              WriteAsiDir=>_."ASiGW-MCC001-bw200-C1: Output"."Dir D1.4.1");
	    
	END_REGION
	
	REGION D1.5.1
	    //D1.5.1
	    #"D1.5.1"(ConveyorID := _."D1.5.1",
	              ConveyorSensor:=_."ASiGW-MCC001-bw200-C1: Input"."Sensor D1.5.1",
	              Fault := DB_UDI.ProductionLine.Fault.Stop.Conveyor[_."D1.5.1"],
	              Upstream := DB_UDI.ProductionLine.Upstream.Conveyor[_."D1.5.1"],
	              Downstream := DB_UDI.ProductionLine.DownstreamAccu.Stop.Conveyor[_."D1.5.1"],
	              Interlock := DB_UDI.ProductionLine.Interlock.Stop.Conveyor[_."D1.5.1"],
	              RunForward=>_."ASiGW-MCC001-bw200-C1: Output"."Motor - D1.5.1",
	              WriteAsiDir=>_."ASiGW-MCC001-bw200-C1: Output"."1-4A Dir",
	              WriteAsiSpeed=>_."ASiGW-MCC001-bw200-C1: Output"."1-4A Speed");
	    
	END_REGION
	
	REGION D1.6.1
	    //D1.6.1
	    #"D1.6.1"(ConveyorID := _."D1.6.1",
	              ConveyorSensor:=_."ASiGW-MCC001-bw200-C1: Input"."Sensor D1.6.1",
	              Fault := DB_UDI.ProductionLine.Fault.Stop.Conveyor[_."D1.6.1"],
	              Upstream := DB_UDI.ProductionLine.Upstream.Conveyor[_."D1.6.1"],
	              Downstream := DB_UDI.ProductionLine.DownstreamAccu.Stop.Conveyor[_."D1.6.1"],
	              Interlock := DB_UDI.ProductionLine.Interlock.Stop.Conveyor[_."D1.6.1"],
	              RunForward=>_."ASiGW-MCC001-bw200-C1: Output"."Motor D1.6.1",
	              WriteAsiDir=>_."ASiGW-MCC001-bw200-C1: Output"."Dir D1.6.1");
	    
	END_REGION
	
	REGION D1.7.1
	    //D1.7.1
	    #"D1.7.1"(ConveyorID := _."D1.7.1",
	              ConveyorSensor:=_."ASiGW-MCC001-bw200-C1: Input"."Sensor D1.7.10",
	              Fault := DB_UDI.ProductionLine.Fault.Stop.Conveyor[_."D1.7.1"],
	              Upstream := DB_UDI.ProductionLine.Upstream.Conveyor[_."D1.7.1"],
	              Downstream := DB_UDI.ProductionLine.DownstreamAccu.Stop.Conveyor[_."D1.7.1"],
	              Interlock := DB_UDI.ProductionLine.Interlock.Stop.Conveyor[_."D1.7.1"],
	              RunForward=>_."ASiGW-MCC001-bw200-C1: Output"."Motor D1.7.1",
	              WriteAsiDir=>_."ASiGW-MCC001-bw200-C1: Output"."Dir D1.7.1");
	    
	END_REGION
	
	REGION D1.7.2
	    //D1.7.2
	    #"D1.7.2"(ConveyorID := _."D1.7.2",
	              ConveyorSensor:=_."ASiGW-MCC001-bw200-C1: Input"."Sensor D1.7.10",
	              Fault := DB_UDI.ProductionLine.Fault.Stop.Conveyor[_."D1.7.2"],
	              Upstream := DB_UDI.ProductionLine.Upstream.Conveyor[_."D1.7.2"],
	              Downstream := DB_UDI.ProductionLine.DownstreamAccu.Stop.Conveyor[_."D1.7.2"],
	              Interlock := DB_UDI.ProductionLine.Interlock.Stop.Conveyor[_."D1.7.2"],
	              RunForward=>_."ASiGW-MCC001-bw200-C1: Output"."Motor D1.7.2",
	              WriteAsiDir=>_."ASiGW-MCC001-bw200-C1: Output"."Dir D1.7.2");
	    
	END_REGION
	
	REGION D1.7.3
	    //D1.7.3
	    #"D1.7.3"(ConveyorID := _."D1.7.3",
	              ConveyorSensor:=_."ASiGW-MCC001-bw200-C1: Input"."Sensor D1.7.10",
	              Fault := DB_UDI.ProductionLine.Fault.Stop.Conveyor[_."D1.7.3"],
	              Upstream := DB_UDI.ProductionLine.Upstream.Conveyor[_."D1.7.3"],
	              Downstream := DB_UDI.ProductionLine.DownstreamAccu.Stop.Conveyor[_."D1.7.3"],
	              Interlock := DB_UDI.ProductionLine.Interlock.Stop.Conveyor[_."D1.7.3"],
	              RunForward=>_."ASiGW-MCC001-bw200-C1: Output"."Motor D1.7.3",
	              WriteAsiDir=>_."ASiGW-MCC001-bw200-C1: Output"."Dir D1.7.3");
	    
	END_REGION
	
	REGION D1.7.4
	    //D1.7.4
	    #"D1.7.4"(ConveyorID := _."D1.7.4",
	              ConveyorSensor:=_."ASiGW-MCC001-bw200-C1: Input"."Sensor D1.7.10",
	              Fault := DB_UDI.ProductionLine.Fault.Stop.Conveyor[_."D1.7.4"],
	              Upstream := DB_UDI.ProductionLine.Upstream.Conveyor[_."D1.7.4"],
	              Downstream := DB_UDI.ProductionLine.DownstreamAccu.Stop.Conveyor[_."D1.7.4"],
	              Interlock := DB_UDI.ProductionLine.Interlock.Stop.Conveyor[_."D1.7.4"],
	              RunForward=>_."ASiGW-MCC001-bw200-C1: Output"."Motor D1.7.4",
	              WriteAsiDir=>_."ASiGW-MCC001-bw200-C1: Output"."Dir D1.7.4");
	    
	END_REGION
	
	REGION D1.7.5
	    //D1.7.5
	    #"D1.7.5"(ConveyorID := _."D1.7.5",
	              ConveyorSensor:=_."ASiGW-MCC001-bw200-C1: Input"."Sensor D1.7.10",
	              Fault := DB_UDI.ProductionLine.Fault.Stop.Conveyor[_."D1.7.5"],
	              Upstream := DB_UDI.ProductionLine.Upstream.Conveyor[_."D1.7.5"],
	              Downstream := DB_UDI.ProductionLine.DownstreamAccu.Stop.Conveyor[_."D1.7.5"],
	              Interlock := DB_UDI.ProductionLine.Interlock.Stop.Conveyor[_."D1.7.5"],
	              RunForward=>_."ASiGW-MCC001-bw200-C1: Output"."Motor D1.7.5",
	              WriteAsiDir=>_."ASiGW-MCC001-bw200-C1: Output"."Dir D1.7.5");
	    
	END_REGION
	
	REGION D1.7.6
	    //D1.7.6
	    #"D1.7.6"(ConveyorID := _."D1.7.6",
	              ConveyorSensor:=_."ASiGW-MCC001-bw200-C1: Input"."Sensor D1.7.10",
	              Fault := DB_UDI.ProductionLine.Fault.Stop.Conveyor[_."D1.7.6"],
	              Upstream := DB_UDI.ProductionLine.Upstream.Conveyor[_."D1.7.6"],
	              Downstream := DB_UDI.ProductionLine.DownstreamAccu.Stop.Conveyor[_."D1.7.6"],
	              Interlock := DB_UDI.ProductionLine.Interlock.Stop.Conveyor[_."D1.7.6"],
	              RunForward=>_."ASiGW-MCC001-bw200-C1: Output"."Motor D1.7.6",
	              WriteAsiDir=>_."ASiGW-MCC001-bw200-C1: Output"."Dir D1.7.6");
	    
	END_REGION
	
	REGION D1.7.7
	    //D1.7.7
	    #"D1.7.7"(ConveyorID := _."D1.7.7",
	              ConveyorSensor:=_."ASiGW-MCC001-bw200-C1: Input"."Sensor D1.7.10",
	              Fault := DB_UDI.ProductionLine.Fault.Stop.Conveyor[_."D1.7.7"],
	              Upstream := DB_UDI.ProductionLine.Upstream.Conveyor[_."D1.7.7"],
	              Downstream := DB_UDI.ProductionLine.DownstreamAccu.Stop.Conveyor[_."D1.7.7"],
	              Interlock := DB_UDI.ProductionLine.Interlock.Stop.Conveyor[_."D1.7.7"],
	              RunForward => _."ASiGW-MCC001-bw200-C1: Output"."Motor D1.7.7",
	              WriteAsiDir => _."ASiGW-MCC001-bw200-C1: Output"."Dir D1.7.7");
	    
	END_REGION
	
	REGION D1.7.8
	    //D1.7.8
	    #"D1.7.8"(ConveyorID := _."D1.7.8",
	              ConveyorSensor:=_."ASiGW-MCC001-bw200-C1: Input"."Sensor D1.7.10",
	              Fault := DB_UDI.ProductionLine.Fault.Stop.Conveyor[_."D1.7.8"],
	              Upstream := DB_UDI.ProductionLine.Upstream.Conveyor[_."D1.7.8"],
	              Downstream := DB_UDI.ProductionLine.DownstreamAccu.Stop.Conveyor[_."D1.7.8"],
	              Interlock := DB_UDI.ProductionLine.Interlock.Stop.Conveyor[_."D1.7.8"],
	              RunForward=>_."ASiGW-MCC001-bw200-C1: Output"."Motor D1.7.8",
	              WriteAsiDir=>_."ASiGW-MCC001-bw200-C1: Output"."Dir D1.7.8");
	    
	END_REGION
	
	REGION D1.7.9
	    //D1.7.9
	    #"D1.7.9"(ConveyorID := _."D1.7.9",
	              ConveyorSensor:=_."ASiGW-MCC001-bw200-C1: Input"."Sensor D1.7.10",
	               Fault := DB_UDI.ProductionLine.Fault.Stop.Conveyor[_."D1.7.9"],
	               Upstream := DB_UDI.ProductionLine.Upstream.Conveyor[_."D1.7.9"],
	               Downstream := DB_UDI.ProductionLine.DownstreamAccu.Stop.Conveyor[_."D1.7.9"],
	               Interlock := DB_UDI.ProductionLine.Interlock.Stop.Conveyor[_."D1.7.9"],
	               RunForward=>_."ASiGW-MCC001-bw200-C1: Output"."Motor D1.7.9",
	               WriteAsiDir=>_."ASiGW-MCC001-bw200-C1: Output"."Dir D1.7.9");
	     
	END_REGION
	
	REGION D1.7.10
	    //D1.7.10
	    #"D1.7.10"(ConveyorID := _."D1.7.10",
	               ConveyorSensor:=_."ASiGW-MCC001-bw200-C1: Input"."Sensor D1.7.10",
	               Fault := DB_UDI.ProductionLine.Fault.Stop.Conveyor[_."D1.7.10"],
	               Upstream := DB_UDI.ProductionLine.Upstream.Conveyor[_."D1.7.10"],
	               Downstream := DB_UDI.ProductionLine.DownstreamAccu.Stop.Conveyor[_."D1.7.10"],
	               Interlock := DB_UDI.ProductionLine.Interlock.Stop.Conveyor[_."D1.7.10"],
	               RunForward => _."ASiGW-MCC001-bw200-C1: Output"."Motor D1.7.10",
	               WriteAsiDir => _."ASiGW-MCC001-bw200-C1: Output"."Dir D1.7.10");
	    
	END_REGION
	
	REGION D1.8.1
	    //D1.8.1
	    #"D1.8.1"(ConveyorID := _."D1.8.1",
	              ConveyorSensor:=_."ASiGW-MCC001-bw200-C1: Input"."Sensor D1.8.1",
	              Fault := DB_UDI.ProductionLine.Fault.Stop.Conveyor[_."D1.8.1"],
	              Upstream := DB_UDI.ProductionLine.Upstream.Conveyor[_."D1.8.1"],
	              Downstream := DB_UDI.ProductionLine.DownstreamAccu.Stop.Conveyor[_."D1.8.1"],
	              Interlock := DB_UDI.ProductionLine.Interlock.Stop.Conveyor[_."D1.8.1"],
	              RunForward => _."ASiGW-MCC001-bw200-C1: Output"."Motor D1.8.1",
	              WriteAsiDir => _."ASiGW-MCC001-bw200-C1: Output"."Dir D1.8.1");
	    
	END_REGION
	
	REGION D1.8.2
	    //D1.8.2
	    #"D1.8.2"(ConveyorID := _."D1.8.2",
	              ConveyorSensor:=_."ASiGW-MCC001-bw200-C1: Input"."Sensor D1.8.2",
	              Fault := DB_UDI.ProductionLine.Fault.Stop.Conveyor[_."D1.8.2"],
	              Upstream := DB_UDI.ProductionLine.Upstream.Conveyor[_."D1.8.2"],
	              Downstream := DB_UDI.ProductionLine.DownstreamAccu.Stop.Conveyor[_."D1.8.2"],
	              Interlock := DB_UDI.ProductionLine.Interlock.Stop.Conveyor[_."D1.8.2"],
	              RunForward => _."ASiGW-MCC001-bw200-C1: Output"."Motor D1.8.2",
	              WriteAsiDir => _."ASiGW-MCC001-bw200-C1: Output"."Dir D1.8.2");
	    
	END_REGION
	
	REGION D1.8.3
	    //D1.8.3
	    #"D1.8.3"(ConveyorID := _."D1.8.3",
	              ConveyorSensor:=_."ASiGW-MCC001-bw200-C1: Input"."Sensor D1.8.3",
	              Fault := DB_UDI.ProductionLine.Fault.Stop.Conveyor[_."D1.8.3"],
	              Upstream := DB_UDI.ProductionLine.Upstream.Conveyor[_."D1.8.3"],
	              Downstream := DB_UDI.ProductionLine.DownstreamAccu.Stop.Conveyor[_."D1.8.3"],
	              Interlock := DB_UDI.ProductionLine.Interlock.Stop.Conveyor[_."D1.8.3"],
	              RunForward => _."ASiGW-MCC001-bw200-C1: Output"."Motor D1.8.3",
	              WriteAsiDir => _."ASiGW-MCC001-bw200-C1: Output"."Dir D1.8.3");
	    
	END_REGION
	
	REGION D1.9.1 Transfer Unit
	    ////Transfer D1.9.1
	    #"D1.9.2"(TransferID := _."D1.9.1",
	              TransferSensor:=_."ASiGW-MCC001-bw200-C1: Input"."LoadPresence -D1.9.1",
	              Fault := DB_UDI.ProductionLine.Fault.Stop.Conveyor[_."D1.9.1"],
	              Upstream := DB_UDI.ProductionLine.Upstream.Conveyor[_."D1.9.1"],
	              FrontSensor:=_."ASiGW-MCC001-bw200-C1: Input"."FrontSensor -D1.9.1",
	              EndSensor:=_."ASiGW-MCC001-bw200-C1: Input"."EndSensor -D1.9.1",
	              "Left/RightSensor":=_."ASiGW-MCC001-bw200-C1: Input"."LeftSensor -D1.9.1",
	              Downstream := DB_UDI.ProductionLine.DownstreamAccu.Stop.Conveyor[_."D1.9.1"],
	              TransferDirection := DB_ToteTracking.Conveyor[_."D1.9.1"].ToteDir,
	              StartSignal => _."ASiGW-MCC001-bw200-C1: Output"."StartSignal -D1.9.1",
	              Cmd1 =>  _."ASiGW-MCC001-bw200-C1: Output"."Command1 -D1.9.1",
	              Cmd2 => _."ASiGW-MCC001-bw200-C1: Output"."Command2 -D1.9.1",
	              ErrorReset =>  _."ASiGW-MCC001-bw200-C1: Output"."ErrorReset -D1.9.1");
	    
	END_REGION
	
	REGION D1.10.1 Transfer Unit
	    ////Transfer D1.10.1
	    #"D1.10.1"(TransferID := _."D1.10.1",
	              Fault := DB_UDI.ProductionLine.Fault.Stop.Conveyor[_."D1.10.1"],
	              Upstream := DB_UDI.ProductionLine.Upstream.Conveyor[_."D1.10.1"],
	              Downstream := DB_UDI.ProductionLine.DownstreamAccu.Stop.Conveyor[_."D1.10.1"],
	              TransferDirection := DB_ToteTracking.Conveyor[_."D1.10.1"].ToteDir,
	              StartSignal =>  _."ASiGW-MCC001-bw200-C1: Output"."StartSignal -D1.10.1",
	              Cmd1 =>  _."ASiGW-MCC001-bw200-C1: Output"."Command1 -D1.10.1",
	              Cmd2 =>  _."ASiGW-MCC001-bw200-C1: Output"."Command2 -D1.10.1",
	              ErrorReset =>  _."ASiGW-MCC001-bw200-C1: Output"."ErrorReset -D1.10.1");
	    
	END_REGION
	
	REGION D1.11.1
	    //D1.11.1
	    #"D1.11.1"(ConveyorID := _."D1.11.1",
	               ConveyorSensor:=_."ASiGW-MCC001-bw200-C1: Input"."Sensor D1.11.1",
	               Fault := DB_UDI.ProductionLine.Fault.Stop.Conveyor[_."D1.11.1"],
	               Upstream := DB_UDI.ProductionLine.Upstream.Conveyor[_."D1.11.1"],
	               Downstream := DB_UDI.ProductionLine.DownstreamAccu.Stop.Conveyor[_."D1.11.1"],
	               Interlock := DB_UDI.ProductionLine.Interlock.Stop.Conveyor[_."D1.11.1"],
	               RunForward => _."ASiGW-MCC001-bw200-C1: Output"."Motor D1.11.1",
	               WriteAsiDir => _."ASiGW-MCC001-bw200-C1: Output"."Dir D1.11.1");
	    
	END_REGION
	
	REGION D1.11.2
	    //D1.11.2
	    #"D1.11.2"(ConveyorID := _."D1.11.2",
	               ConveyorSensor:=_."ASiGW-MCC001-bw200-C1: Input"."Sensor D1.11.2",
	               Fault := DB_UDI.ProductionLine.Fault.Stop.Conveyor[_."D1.11.2"],
	               Upstream := DB_UDI.ProductionLine.Upstream.Conveyor[_."D1.11.2"],
	               Downstream := DB_UDI.ProductionLine.DownstreamAccu.Stop.Conveyor[_."D1.11.2"],
	               Interlock := DB_UDI.ProductionLine.Interlock.Stop.Conveyor[_."D1.11.2"],
	               RunForward => _."ASiGW-MCC001-bw200-C1: Output"."Motor D1.11.2",
	               WriteAsiDir => _."ASiGW-MCC001-bw200-C1: Output"."Dir D1.11.2");
	    
	END_REGION
	
	REGION D1.11.3
	    //D1.11.3
	    #"D1.11.3"(ConveyorID := _."D1.11.3",
	               ConveyorSensor:=_."ASiGW-MCC001-bw200-C1: Input"."Sensor D1.11.3",
	               Fault := DB_UDI.ProductionLine.Fault.Stop.Conveyor[_."D1.11.3"],
	               Upstream := DB_UDI.ProductionLine.Upstream.Conveyor[_."D1.11.3"],
	               Downstream := DB_UDI.ProductionLine.DownstreamAccu.Stop.Conveyor[_."D1.11.3"],
	               Interlock := DB_UDI.ProductionLine.Interlock.Stop.Conveyor[_."D1.11.3"],
	               RunForward => _."ASiGW-MCC001-bw200-C1: Output"."Motor D1.11.3",
	               WriteAsiDir => _."ASiGW-MCC001-bw200-C1: Output"."Dir D1.11.3");
	    
	END_REGION
	
	REGION D1.12.1
	    //D1.12.1
	    #"D1.12.1"(ConveyorID := _."D1.12.1",
	               ConveyorSensor:=_."ASiGW-MCC001-bw200-C1: Input"."Sensor D1.12.3",
	               Fault := DB_UDI.ProductionLine.Fault.Stop.Conveyor[_."D1.12.1"],
	               Upstream := DB_UDI.ProductionLine.Upstream.Conveyor[_."D1.12.1"],
	               Downstream := DB_UDI.ProductionLine.DownstreamAccu.Stop.Conveyor[_."D1.12.1"],
	               Interlock := DB_UDI.ProductionLine.Interlock.Stop.Conveyor[_."D1.12.1"],
	               RunForward=>_."ASiGW-MCC001-bw200-C1: Output"."Motor D1.12.1",
	               WriteAsiDir=>_."ASiGW-MCC001-bw200-C1: Output"."Dir D1.12.1");
	    
	END_REGION
	
	REGION D1.12.2
	    //D1.12.2
	    #"D1.12.2"(ConveyorID := _."D1.12.2",
	               ConveyorSensor:=_."ASiGW-MCC001-bw200-C1: Input"."Sensor D1.12.3",
	               Fault := DB_UDI.ProductionLine.Fault.Stop.Conveyor[_."D1.12.2"],
	               Upstream := DB_UDI.ProductionLine.Upstream.Conveyor[_."D1.12.2"],
	               Downstream := DB_UDI.ProductionLine.DownstreamAccu.Stop.Conveyor[_."D1.12.2"],
	               Interlock := DB_UDI.ProductionLine.Interlock.Stop.Conveyor[_."D1.12.2"],
	               RunForward => _."ASiGW-MCC001-bw200-C1: Output"."Motor D1.12.2",
	               WriteAsiDir => _."ASiGW-MCC001-bw200-C1: Output"."Dir D1.12.2");
	    
	END_REGION
	
	REGION D1.12.3
	    ////End
	    #"D1.12.3"(ConveyorID := _."D1.12.3",
	               ConveyorSensor:=_."ASiGW-MCC001-bw200-C1: Input"."Sensor D1.12.3",
	               Fault := DB_UDI.ProductionLine.Fault.Stop.Conveyor[_."D1.12.3"],
	               Upstream := DB_UDI.ProductionLine.Upstream.Conveyor[_."D1.12.3"],
	               Downstream := DB_UDI.ProductionLine.DownstreamAccu.Stop.Conveyor[_."D1.12.3"],
	               Interlock := DB_UDI.ProductionLine.Interlock.Stop.Conveyor[_."D1.12.3"],
	               RunForward => _."ASiGW-MCC001-bw200-C1: Output"."Motor D1.12.3",
	               WriteAsiDir => _."ASiGW-MCC001-bw200-C1: Output"."Dir D1.12.3");
	    
	END_REGION
	
	REGION E1.1.1
	    //E1.1.1
	    #"E1.1.1"(ConveyorID := _."E1.1.1",
	              ConveyorSensor:=_."ASiGW-MCC001-bw200-C1: Input"."Sensor E1.1.1",
	              Fault := DB_UDI.ProductionLine.Fault.Stop.Conveyor[_."E1.1.1"],
	              Upstream := DB_UDI.ProductionLine.Upstream.Conveyor[_."E1.1.1"],
	              Downstream := DB_UDI.ProductionLine.DownstreamAccu.Stop.Conveyor[_."E1.1.1"],
	              Interlock := DB_UDI.ProductionLine.Interlock.Stop.Conveyor[_."E1.1.1"],
	              RunForward=>_."ASiGW-MCC001-bw200-C1: Output"."Motor E1.1.1",
	              WriteAsiDir=>_."ASiGW-MCC001-bw200-C1: Output"."Dir E1.1.1");
	    
	END_REGION
	
	REGION E1.1.2
	    //E1.1.2
	    #"E1.1.2"(ConveyorID := _."E1.1.2",
	              ConveyorSensor:=_."ASiGW-MCC001-bw200-C1: Input"."Sensor E1.1.4",
	              Fault := DB_UDI.ProductionLine.Fault.Stop.Conveyor[_."E1.1.2"],
	              Upstream := DB_UDI.ProductionLine.Upstream.Conveyor[_."E1.1.2"],
	              Downstream := DB_UDI.ProductionLine.DownstreamAccu.Stop.Conveyor[_."E1.1.2"],
	              Interlock := DB_UDI.ProductionLine.Interlock.Stop.Conveyor[_."E1.1.2"],
	              RunForward=>_."ASiGW-MCC001-bw200-C1: Output"."Motor E1.1.2",
	              WriteAsiDir=>_."ASiGW-MCC001-bw200-C1: Output"."Dir E1.1.2");
	    
	END_REGION
	
	REGION E1.1.3
	    //E1.1.3
	    #"E1.1.3"(ConveyorID := _."E1.1.3",
	              ConveyorSensor:=_."ASiGW-MCC001-bw200-C1: Input"."Sensor E1.1.4",
	              Fault := DB_UDI.ProductionLine.Fault.Stop.Conveyor[_."E1.1.3"],
	              Upstream := DB_UDI.ProductionLine.Upstream.Conveyor[_."E1.1.3"],
	              Downstream := DB_UDI.ProductionLine.DownstreamAccu.Stop.Conveyor[_."E1.1.3"],
	              Interlock := DB_UDI.ProductionLine.Interlock.Stop.Conveyor[_."E1.1.3"],
	              RunForward=>_."ASiGW-MCC001-bw200-C1: Output"."Motor E1.1.3",
	              WriteAsiDir=>_."ASiGW-MCC001-bw200-C1: Output"."Dir E1.1.3");
	    
	END_REGION
	
	REGION E1.1.4
	    //E1.1.4
	    #"E1.1.4"(ConveyorID := _."E1.1.4",
	              ConveyorSensor:=_."ASiGW-MCC001-bw200-C1: Input"."Sensor E1.1.4",
	              Fault := DB_UDI.ProductionLine.Fault.Stop.Conveyor[_."E1.1.4"],
	              Upstream := DB_UDI.ProductionLine.Upstream.Conveyor[_."E1.1.4"],
	              Downstream := DB_UDI.ProductionLine.DownstreamAccu.Stop.Conveyor[_."E1.1.4"],
	              Interlock := DB_UDI.ProductionLine.Interlock.Stop.Conveyor[_."E1.1.4"],
	              RunForward=>_."ASiGW-MCC001-bw200-C1: Output"."Motor E1.1.4",
	              WriteAsiDir=>_."ASiGW-MCC001-bw200-C1: Output"."Dir E1.1.4");
	    
	END_REGION
	
	REGION E1.2.1
	    //E1.2.1
	    #"E1.2.1"(ConveyorID := _."E1.2.1",
	              ConveyorSensor:=_."ASiGW-MCC001-bw200-C1: Input"."Sensor E1.2.1",
	              Fault := DB_UDI.ProductionLine.Fault.Stop.Conveyor[_."E1.2.1"],
	              Upstream := DB_UDI.ProductionLine.Upstream.Conveyor[_."E1.2.1"],
	              Downstream := DB_UDI.ProductionLine.DownstreamAccu.Stop.Conveyor[_."E1.2.1"],
	              Interlock := DB_UDI.ProductionLine.Interlock.Stop.Conveyor[_."E1.2.1"],
	              RunForward=>_."ASiGW-MCC001-bw200-C1: Output"."Motor - E1.2.1",
	              WriteAsiDir=>_."ASiGW-MCC001-bw200-C1: Output"."1-21A Dir",
	              WriteAsiSpeed=>_."ASiGW-MCC001-bw200-C1: Output"."1-21A Speed");
	    
	END_REGION
	
	REGION E1.3.1
	    //E1.3.1
	    #"E1.3.1"(ConveyorID := _."E1.3.1",
	              ConveyorSensor:=_."ASiGW-MCC001-bw200-C1: Input"."Sensor E1.3.1",
	              Fault := DB_UDI.ProductionLine.Fault.Stop.Conveyor[_."E1.3.1"],
	              Upstream := DB_UDI.ProductionLine.Upstream.Conveyor[_."E1.3.1"],
	              Downstream := DB_UDI.ProductionLine.DownstreamAccu.Stop.Conveyor[_."E1.3.1"],
	              Interlock := DB_UDI.ProductionLine.Interlock.Stop.Conveyor[_."E1.3.1"],
	              RunForward=>_."ASiGW-MCC001-bw200-C1: Output"."Motor - E1.3.1",
	              WriteAsiDir=>_."ASiGW-MCC001-bw200-C1: Output"."1-21A Dir",
	              WriteAsiSpeed=>_."ASiGW-MCC001-bw200-C1: Output"."1-21A Speed");
	    
	END_REGION
	
	REGION E1.4.1
	    //E1.4.1
	    #"E1.4.1"(ConveyorID := _."E1.4.1",
	              ConveyorSensor:=_."ASiGW-MCC001-bw200-C1: Input"."Sensor E1.4.1",
	              Fault := DB_UDI.ProductionLine.Fault.Stop.Conveyor[_."E1.4.1"],
	              Upstream := DB_UDI.ProductionLine.Upstream.Conveyor[_."E1.4.1"],
	              Downstream := DB_UDI.ProductionLine.DownstreamAccu.Stop.Conveyor[_."E1.4.1"],
	              Interlock := DB_UDI.ProductionLine.Interlock.Stop.Conveyor[_."E1.4.1"],
	              RunForward=>_."ASiGW-MCC001-bw200-C1: Output"."Motor E1.4.1",
	              WriteAsiDir=>_."ASiGW-MCC001-bw200-C1: Output"."Dir E1.4.1");
	    
	END_REGION
	
	REGION E1.5.1
	    //E1.5.1
	    #"E1.5.1"(ConveyorID := _."E1.5.1",
	              ConveyorSensor := _."ASiGW-MCC001-bw200-C1: Input"."Sensor E1.5.1",
	              Fault := DB_UDI.ProductionLine.Fault.Stop.Conveyor[_."E1.5.1"],
	              Upstream := DB_UDI.ProductionLine.Upstream.Conveyor[_."E1.5.1"],
	              Downstream := DB_UDI.ProductionLine.DownstreamAccu.Stop.Conveyor[_."E1.5.1"],
	              Interlock := DB_UDI.ProductionLine.Interlock.Stop.Conveyor[_."E1.5.1"],
	              RunForward => _."ASiGW-MCC001-bw200-C1: Output"."Motor - E1.5.1",
	              WriteAsiDir => _."ASiGW-MCC001-bw200-C1: Output"."1-23A Dir",
	              WriteAsiSpeed => _."ASiGW-MCC001-bw200-C1: Output"."1-23A Speed");
	    
	    
	END_REGION
	
	REGION E1.6.1
	    ////E1.6.1 Arm for Merger2
	    #"E1.6.1"(ConveyorID := _."E1.6.1",
	              ConveyorSensor:=_."ASiGW-MCC001-bw200-C1: Input"."Sensor E1.5.1",
	              Fault := DB_UDI.ProductionLine.Fault.Stop.Conveyor[_."E1.6.1"],
	              Upstream := DB_UDI.ProductionLine.Upstream.Conveyor[_."E1.6.1"],
	              Downstream := DB_UDI.ProductionLine.DownstreamAccu.Stop.Conveyor[_."E1.6.1"],
	              Interlock := DB_UDI.ProductionLine.Interlock.Stop.Conveyor[_."E1.6.1"],
	              RunForward=>_."ASiGW-MCC001-bw200-C1: Output"."Motor E1.6.1",
	              WriteAsiDir=>_."ASiGW-MCC001-bw200-C1: Output"."Dir E1.6.1");
	    
	END_REGION
	
	
END_FUNCTION_BLOCK
END_NAMESPACE

NAMESPACE ProductionLine
ORGANIZATION_BLOCK Main_ProductionLine
TITLE = "Main Program Sweep (Cycle)"
{ S7_Optimized_Access := 'TRUE' ; Published := 'FALSE' }
VERSION : 0.1

BEGIN
	// ==========================================================================================================================================
	// Company        : LogTech, s.r.o.
	// Created by     : Mahmoud Elnady
	// Block          : FB_Main_LineA1
	// Project        : Lékárna Chrudim
	// Project number : 23-157
	// ==========================================================================================================================================
	
	
	//Synchronization Line_A1 and Global
	
	REGION Synchronization
	    
	    FC_Sync();
	    
	END_REGION
	
	REGION Line A1
	    
	    IDB_ProductionLine();
	    
	    //Upstream
	    FC_Upstream();
	    
	    //Downstream
	    FC_Downstream();
	    
	    //Fault
	    FC_Fault();
	    
	    // Merging
	    IDB_Merging();
	    
	    // Barcode
	    IDB_BarcodeReader();
	    
	    // OPC Server
	    IDB_OPC_Communication();
	    
	    //FB Technology
	    IDB_FB_Technology();
	    
	    //Tote Tracking
	    IDB_ToteTracking();
	    
	    // FB Segments Status
	    IDB_Segments_Status();
	    
	    // FB Toggle Dir
	    IDB_FB_ToggleDir();
	
	END_REGION
	
	REGION Test
	    // Flow Test
	    IDB_Flow_Test();
	    
	END_REGION
	
	
	
	
	
	
	
	
	
	
	
	
END_ORGANIZATION_BLOCK
END_NAMESPACE

NAMESPACE EmptyLine
FUNCTION FC_Init : Void
{ S7_Optimized_Access := 'TRUE' ; Published := 'TRUE' }
VERSION : 0.1

BEGIN
	// ==========================================================================================================================================
	// Company        : LogTech, s.r.o.
	// Created by     : Anton Vinoth Soundraraj
	// Block          : FC_Init
	// Project        : Lékarna DC Chrudim
	// Project number : 23-157
	// ==========================================================================================================================================
	
	
	
	
	
	
	
	
	
	
	
	
	
	
	
END_FUNCTION
END_NAMESPACE

NAMESPACE EmptyLine
FUNCTION_BLOCK FB_Interlock
{ S7_Optimized_Access := 'TRUE' ; Published := 'TRUE' }
VERSION : 0.1
   VAR 
      "J1.2.3" : _.Global.FB_Interlock;
      "J2.3.1" : _.Global.FB_Interlock;
      "J1.5.4_Straight" : _.Global.FB_Interlock;
      "J1.5.4_Left" : _.Global.FB_Interlock;
      "InterlockJ1.7.1" { S7_SetPoint := 'True'} : Bool;
      "InterlockK1.2.1" : Bool;
   END_VAR


BEGIN
	// ==========================================================================================================================================
	// Company        : LogTech, s.r.o.
	// Created by     : Anton Vinoth Soundraraj
	// Block          : FB_Interlock
	// Project        : Lékarna DC Chrudim
	// Project number : 23-157
	// ==========================================================================================================================================
	
	REGION J1.2.3
	    // J1.2.3
	    #"J1.2.3"(ConveyorSensor := IDB_EmptyLine."J1.2.3".FilteredSensor,
	              DownstreamOccuTime := DB_ConveyorParameters.Line.EmptyLine.Conveyor[_."J2.1.4"].ConvOccTime,
	              StopConv => DB_UDI.EmptyLine.Interlock.Stop.Conveyor[_."J2.1.3"]);
	    
	END_REGION
	
	REGION J2.3.1
	    // J2.3.1
	    #"J2.3.1"(ConveyorSensor := IDB_EmptyLine."J2.3.1".FilteredSensor,
	              DownstreamOccuTime := DB_ConveyorParameters.Line.EmptyLine.Conveyor[_."J2.1.4"].ConvOccTime,
	              StopConv => DB_UDI.EmptyLine.Interlock.Stop.Conveyor[_."J2.3.1"]);
	    
	END_REGION
	
	REGION J1.5.4
	    // J1.5.4
	    #"J1.5.4_Straight"(ConveyorSensor := IDB_EmptyLine."J1.2.5".FilteredSensor AND
	                       ToteDir.Conveyor[_."J1.6.1"].Straight AND
	                       ToteDir.Conveyor[_."J1.6.2"].Straight,
	                       DownstreamOccuTime := DB_ConveyorParameters.Line.EmptyLine.Conveyor[_."J1.7.1"].ConvOccTime,
	                       StopConv => #"InterlockJ1.7.1");
	    
	    #"J1.5.4_Left"(ConveyorSensor := IDB_EmptyLine."J1.2.5".FilteredSensor AND
	                   ToteDir.Conveyor[_."J1.6.1"].toLeft AND
	                   ToteDir.Conveyor[_."J1.6.2"].toLeft,
	                   DownstreamOccuTime := DB_ConveyorParameters.Line.EmptyLine.Conveyor[_."K1.2.1"].ConvOccTime,
	                   StopConv => #"InterlockK1.2.1");
	    
	    
	    DB_UDI.EmptyLine.Interlock.Stop.Conveyor[_."J1.2.5"] := #"InterlockJ1.7.1" OR #"InterlockK1.2.1";
	    
	END_REGION
	
	
	
	
	
	
	
	
	
	
END_FUNCTION_BLOCK
END_NAMESPACE

NAMESPACE EmptyLine
FUNCTION FC_Downstream : Void
{ S7_Optimized_Access := 'TRUE' ; Published := 'TRUE' }
VERSION : 0.1

BEGIN
	// ==========================================================================================================================================
	// Company        : LogTech, s.r.o.
	// Created by     : Anton Vinoth Soundraraj
	// Block          : FC_Downstream
	// Project        : Lékarna DC Chrudim
	// Project number : 23-157
	// ==========================================================================================================================================
	
	REGION J1.1.1
	    //J1.1.1
	    DB_UDI.EmptyLine.DownstreamAcu.Stop.Conveyor[_."J1.1.1"] :=
	    IDB_EmptyLine."J1.1.2".FilteredSensor OR
	    NOT IDB_EmptyLine."J1.1.2".ReadConveyorStatus.ReadytoRun;
	    
	END_REGION
	
	REGION J1.1.2
	    //J1.1.2
	    DB_UDI.EmptyLine.DownstreamAcu.Stop.Conveyor[_."J1.1.2"] :=
	    IDB_EmptyLine."J1.1.11".FilteredSensor OR
	    NOT IDB_EmptyLine."J1.1.3".ReadConveyorStatus.ReadytoRun OR
	    NOT IDB_EmptyLine."J1.1.4".ReadConveyorStatus.ReadytoRun OR
	    NOT IDB_EmptyLine."J1.1.5".ReadConveyorStatus.ReadytoRun OR
	    NOT IDB_EmptyLine."J1.1.6".ReadConveyorStatus.ReadytoRun OR
	    NOT IDB_EmptyLine."J1.1.7".ReadConveyorStatus.ReadytoRun OR
	    NOT IDB_EmptyLine."J1.1.8".ReadConveyorStatus.ReadytoRun OR
	    NOT IDB_EmptyLine."J1.1.9".ReadConveyorStatus.ReadytoRun OR
	    NOT IDB_EmptyLine."J1.1.10".ReadConveyorStatus.ReadytoRun OR
	    NOT IDB_EmptyLine."J1.1.11".ReadConveyorStatus.ReadytoRun;
	    
	END_REGION
	
	REGION J1.1.3 TO J1.1.11 
	    REGION J1.1.3
	        //J1.1.3
	        DB_UDI.EmptyLine.DownstreamAcu.Stop.Conveyor[_."J1.1.3"] :=
	        DB_UDI.EmptyLine.DownstreamAcu.Stop.Conveyor[_."J1.1.4"];
	        
	    END_REGION
	    
	    REGION J1.1.4
	        //J1.1.4
	        DB_UDI.EmptyLine.DownstreamAcu.Stop.Conveyor[_."J1.1.4"] :=
	        DB_UDI.EmptyLine.DownstreamAcu.Stop.Conveyor[_."J1.1.5"];
	        
	    END_REGION
	    
	    REGION J1.1.5
	        //J1.1.5
	        DB_UDI.EmptyLine.DownstreamAcu.Stop.Conveyor[_."J1.1.5"] :=
	        DB_UDI.EmptyLine.DownstreamAcu.Stop.Conveyor[_."J1.1.6"];
	        
	    END_REGION
	    
	    REGION J1.1.6
	        //J1.1.6
	        DB_UDI.EmptyLine.DownstreamAcu.Stop.Conveyor[_."J1.1.6"] :=
	        DB_UDI.EmptyLine.DownstreamAcu.Stop.Conveyor[_."J1.1.7"];
	        
	    END_REGION
	    
	    REGION J1.1.7
	        //J1.1.7
	        DB_UDI.EmptyLine.DownstreamAcu.Stop.Conveyor[_."J1.1.7"] :=
	        DB_UDI.EmptyLine.DownstreamAcu.Stop.Conveyor[_."J1.1.8"];
	        
	    END_REGION
	    
	    REGION J1.1.8
	        //J1.1.8
	        DB_UDI.EmptyLine.DownstreamAcu.Stop.Conveyor[_."J1.1.8"] :=
	        DB_UDI.EmptyLine.DownstreamAcu.Stop.Conveyor[_."J1.1.9"];
	        
	    END_REGION
	    
	    REGION J1.1.9
	        //J1.1.9
	        DB_UDI.EmptyLine.DownstreamAcu.Stop.Conveyor[_."J1.1.9"] :=
	        DB_UDI.EmptyLine.DownstreamAcu.Stop.Conveyor[_."J1.1.10"];
	        
	    END_REGION
	    
	    REGION J1.1.10
	        //J1.1.10
	        DB_UDI.EmptyLine.DownstreamAcu.Stop.Conveyor[_."J1.1.10"] :=
	        DB_UDI.EmptyLine.DownstreamAcu.Stop.Conveyor[_."J1.1.11"];
	        
	    END_REGION
	    
	    REGION J1.1.11
	        //J1.1.11
	        DB_UDI.EmptyLine.DownstreamAcu.Stop.Conveyor[_."J1.1.11"] :=
	        IDB_EmptyLine."J1.1.15".FilteredSensor OR
	        NOT IDB_EmptyLine."J1.1.12".ReadConveyorStatus.ReadytoRun OR
	        NOT IDB_EmptyLine."J1.1.13".ReadConveyorStatus.ReadytoRun OR
	        NOT IDB_EmptyLine."J1.1.14".ReadConveyorStatus.ReadytoRun OR
	        NOT IDB_EmptyLine."J1.1.15".ReadConveyorStatus.ReadytoRun;
	        
	    END_REGION
	END_REGION
	
	
	REGION J1.1.12 TO J1.1.15
	    REGION J1.1.12
	        //J1.1.12
	        DB_UDI.EmptyLine.DownstreamAcu.Stop.Conveyor[_."J1.1.12"] :=
	        DB_UDI.EmptyLine.DownstreamAcu.Stop.Conveyor[_."J1.1.13"];
	        
	    END_REGION
	    
	    REGION J1.1.13
	        //J1.1.13
	        DB_UDI.EmptyLine.DownstreamAcu.Stop.Conveyor[_."J1.1.13"] :=
	        DB_UDI.EmptyLine.DownstreamAcu.Stop.Conveyor[_."J1.1.14"];
	        
	    END_REGION
	    
	    REGION J1.1.14
	        //J1.1.14
	        DB_UDI.EmptyLine.DownstreamAcu.Stop.Conveyor[_."J1.1.14"] :=
	        DB_UDI.EmptyLine.DownstreamAcu.Stop.Conveyor[_."J1.1.15"];
	        
	    END_REGION
	    
	    REGION J1.1.15
	        //J1.1.15
	        DB_UDI.EmptyLine.DownstreamAcu.Stop.Conveyor[_."J1.1.15"] :=
	        IDB_EmptyLine."J1.2.1".FilteredSensor OR
	        NOT IDB_EmptyLine."J1.2.1".ReadConveyorStatus.ReadytoRun;
	        
	    END_REGION
	END_REGION
	
	REGION J1.2.1
	    //J1.2.1
	    DB_UDI.EmptyLine.DownstreamAcu.Stop.Conveyor[_."J1.2.1"] :=
	    IDB_EmptyLine."J1.2.2".FilteredSensor OR
	    NOT IDB_EmptyLine."J1.2.2".ReadConveyorStatus.ReadytoRun;
	    
	END_REGION
	
	REGION J1.2.2
	    //J1.2.2
	    DB_UDI.EmptyLine.DownstreamAcu.Stop.Conveyor[_."J1.2.2"] :=
	    IDB_EmptyLine."J1.2.3".FilteredSensor OR
	    NOT IDB_EmptyLine."J1.2.3".ReadConveyorStatus.ReadytoRun;
	    
	END_REGION
	
	REGION J1.2.3 Staright for Merger1
	    //J1.2.3 Staright for Merger1
	    DB_UDI.EmptyLine.DownstreamAcu.Stop.Conveyor[_."J1.2.3"] :=
	    IDB_EmptyLine."J2.1.1".FilteredSensor OR
	    NOT IDB_EmptyLine."J2.1.1".ReadConveyorStatus.ReadytoRun OR
	    IDB_Merging."Merge_J1.2.4".Priority.Arm OR
	    NOT IDB_Merging."Merge_J1.2.4".Priority.Straight;
	    
	END_REGION
	
	REGION J2.1.1
	    //J2.1.1
	    DB_UDI.EmptyLine.DownstreamAcu.Stop.Conveyor[_."J2.1.1"] :=
	    IDB_EmptyLine."J2.1.2".FilteredSensor OR
	    NOT IDB_EmptyLine."J2.1.2".ReadConveyorStatus.ReadytoRun OR
	    NOT IDB_EmptyLine."J2.1.3".ReadConveyorStatus.ReadytoRun OR
	    NOT IDB_EmptyLine."J2.1.4".ReadConveyorStatus.ReadytoRun OR
	    NOT IDB_EmptyLine."J2.1.5".ReadConveyorStatus.ReadytoRun OR
	    NOT IDB_EmptyLine."J2.1.6".ReadConveyorStatus.ReadytoRun OR
	    NOT IDB_EmptyLine."J2.1.7".ReadConveyorStatus.ReadytoRun OR
	    NOT IDB_EmptyLine."J2.1.8".ReadConveyorStatus.ReadytoRun OR
	    NOT IDB_EmptyLine."J2.1.9".ReadConveyorStatus.ReadytoRun OR
	    NOT IDB_EmptyLine."J2.1.10".ReadConveyorStatus.ReadytoRun OR
	    NOT IDB_EmptyLine."J2.1.11".ReadConveyorStatus.ReadytoRun;
	    
	END_REGION
	
	REGION J2.1.3 TO J2.1.11
	    REGION J2.1.2
	        //J2.1.2
	        DB_UDI.EmptyLine.DownstreamAcu.Stop.Conveyor[_."J2.1.2"] :=
	        DB_UDI.EmptyLine.DownstreamAcu.Stop.Conveyor[_."J2.1.3"];
	        
	    END_REGION
	    
	    REGION J2.1.3
	        //J2.1.3
	        DB_UDI.EmptyLine.DownstreamAcu.Stop.Conveyor[_."J2.1.3"] :=
	        DB_UDI.EmptyLine.DownstreamAcu.Stop.Conveyor[_."J2.1.4"];
	        
	    END_REGION
	    
	    REGION J2.1.4
	        //J2.1.4
	        DB_UDI.EmptyLine.DownstreamAcu.Stop.Conveyor[_."J2.1.4"] :=
	        DB_UDI.EmptyLine.DownstreamAcu.Stop.Conveyor[_."J2.1.5"];
	        
	    END_REGION
	    
	    REGION J2.1.5
	        //J2.1.5
	        DB_UDI.EmptyLine.DownstreamAcu.Stop.Conveyor[_."J2.1.5"] :=
	        DB_UDI.EmptyLine.DownstreamAcu.Stop.Conveyor[_."J2.1.6"];
	        
	    END_REGION
	    
	    REGION J2.1.6
	        //J2.1.6
	        DB_UDI.EmptyLine.DownstreamAcu.Stop.Conveyor[_."J2.1.6"] :=
	        DB_UDI.EmptyLine.DownstreamAcu.Stop.Conveyor[_."J2.1.7"];
	        
	    END_REGION
	    
	    REGION J2.1.7
	        //J2.1.7
	        DB_UDI.EmptyLine.DownstreamAcu.Stop.Conveyor[_."J2.1.7"] :=
	        DB_UDI.EmptyLine.DownstreamAcu.Stop.Conveyor[_."J2.1.8"];
	        
	    END_REGION
	    
	    REGION J2.1.8
	        //J2.1.8
	        DB_UDI.EmptyLine.DownstreamAcu.Stop.Conveyor[_."J2.1.8"] :=
	        DB_UDI.EmptyLine.DownstreamAcu.Stop.Conveyor[_."J2.1.9"];
	        
	    END_REGION
	    
	    REGION J2.1.9
	        //J2.1.9
	        DB_UDI.EmptyLine.DownstreamAcu.Stop.Conveyor[_."J2.1.9"] :=
	        DB_UDI.EmptyLine.DownstreamAcu.Stop.Conveyor[_."J2.1.10"];
	        
	    END_REGION
	    
	    REGION J2.1.10
	        //J2.1.10
	        DB_UDI.EmptyLine.DownstreamAcu.Stop.Conveyor[_."J2.1.10"] :=
	        DB_UDI.EmptyLine.DownstreamAcu.Stop.Conveyor[_."J2.1.11"];
	        
	    END_REGION
	    
	    REGION J2.1.11
	        //J2.1.11
	        DB_UDI.EmptyLine.DownstreamAcu.Stop.Conveyor[_."J2.1.11"] :=
	        IDB_EmptyLine."J2.1.15".FilteredSensor OR
	        NOT IDB_EmptyLine."J2.1.12".ReadConveyorStatus.ReadytoRun OR
	        NOT IDB_EmptyLine."J2.1.13".ReadConveyorStatus.ReadytoRun OR
	        NOT IDB_EmptyLine."J2.1.14".ReadConveyorStatus.ReadytoRun OR
	        NOT IDB_EmptyLine."J2.1.15".ReadConveyorStatus.ReadytoRun;
	        
	    END_REGION
	END_REGION
	
	
	REGION J2.1.12 TO J2.1.15 
	    REGION J2.1.12
	        //J2.1.12
	        DB_UDI.EmptyLine.DownstreamAcu.Stop.Conveyor[_."J2.1.12"] :=
	        DB_UDI.EmptyLine.DownstreamAcu.Stop.Conveyor[_."J2.1.13"];
	        
	    END_REGION
	    
	    REGION J2.1.13
	        //J2.1.13
	        DB_UDI.EmptyLine.DownstreamAcu.Stop.Conveyor[_."J2.1.13"] :=
	        DB_UDI.EmptyLine.DownstreamAcu.Stop.Conveyor[_."J2.1.14"];
	        
	    END_REGION
	    
	    REGION J2.1.14
	        //J2.1.14
	        DB_UDI.EmptyLine.DownstreamAcu.Stop.Conveyor[_."J2.1.14"] :=
	        DB_UDI.EmptyLine.DownstreamAcu.Stop.Conveyor[_."J2.1.15"];
	        
	    END_REGION
	    
	    REGION J2.1.15
	        //J2.1.15
	        DB_UDI.EmptyLine.DownstreamAcu.Stop.Conveyor[_."J2.1.15"] :=
	        IDB_EmptyLine."J2.2.1".FilteredSensor OR
	        NOT IDB_EmptyLine."J2.2.1".ReadConveyorStatus.ReadytoRun;
	        
	    END_REGION
	END_REGION
	
	
	REGION J2.2.1
	    //J2.2.1
	    DB_UDI.EmptyLine.DownstreamAcu.Stop.Conveyor[_."J2.2.1"] :=
	    IDB_EmptyLine."J2.2.2".FilteredSensor OR
	    NOT IDB_EmptyLine."J2.2.2".ReadConveyorStatus.ReadytoRun;
	    
	END_REGION
	
	REGION J2.2.2
	    //J2.2.2
	    DB_UDI.EmptyLine.DownstreamAcu.Stop.Conveyor[_."J2.2.2"] :=
	    IDB_EmptyLine."J2.3.1".FilteredSensor OR
	    NOT IDB_EmptyLine."J2.3.1".ReadConveyorStatus.ReadytoRun;
	    
	END_REGION
	
	REGION J2.3.1 TO J2.4.1 
	    REGION J2.3.1
	        //J2.3.1
	        DB_UDI.EmptyLine.DownstreamAcu.Stop.Conveyor[_."J2.3.1"] :=
	        DB_UDI.EmptyLine.DownstreamAcu.Stop.Conveyor[_."J2.4.1"];
	        
	    END_REGION
	    
	    REGION J2.4.1 Arm for Merger1
	        //J2.4.1 Arm for Merger1
	        DB_UDI.EmptyLine.DownstreamAcu.Stop.Conveyor[_."J2.4.1"] :=
	        IDB_EmptyLine."J1.2.4".FilteredSensor OR
	        NOT IDB_EmptyLine."J1.2.4".ReadConveyorStatus.ReadytoRun OR
	        NOT IDB_Merging."Merge_J1.2.4".Priority.Arm OR
	        IDB_Merging."Merge_J1.2.4".Priority.Straight;
	    END_REGION
	END_REGION
	
	
	REGION J1.2.4 Merger 1
	    //J1.2.4 Merger 1
	    DB_UDI.EmptyLine.DownstreamAcu.Stop.Conveyor[_."J1.2.4"] :=
	    IDB_EmptyLine."J1.2.5".FilteredSensor OR
	    NOT IDB_EmptyLine."J1.2.5".ReadConveyorStatus.ReadytoRun;
	    
	END_REGION
	
	REGION J1.2.5
	    //J1.2.5
	    DB_UDI.EmptyLine.DownstreamAcu.Stop.Conveyor[_."J1.2.5"] :=
	    IDB_EmptyLine."J1.4.7".FilteredSensor OR
	    NOT IDB_EmptyLine."J1.3.1".ReadConveyorStatus.ReadytoRun OR
	    NOT IDB_EmptyLine."J1.3.2".ReadConveyorStatus.ReadytoRun OR
	    NOT IDB_EmptyLine."J1.4.1".ReadConveyorStatus.ReadytoRun OR
	    NOT IDB_EmptyLine."J1.4.2".ReadConveyorStatus.ReadytoRun OR
	    NOT IDB_EmptyLine."J1.4.3".ReadConveyorStatus.ReadytoRun OR
	    NOT IDB_EmptyLine."J1.4.4".ReadConveyorStatus.ReadytoRun OR
	    NOT IDB_EmptyLine."J1.4.5".ReadConveyorStatus.ReadytoRun OR
	    NOT IDB_EmptyLine."J1.4.6".ReadConveyorStatus.ReadytoRun OR
	    NOT IDB_EmptyLine."J1.4.7".ReadConveyorStatus.ReadytoRun OR
	    NOT IDB_EmptyLine."J1.5.1".ReadConveyorStatus.ReadytoRun;
	    
	END_REGION
	
	REGION J1.3.1 TO J1.4.7
	    REGION J1.3.1
	        //J1.3.1
	        DB_UDI.EmptyLine.DownstreamAcu.Stop.Conveyor[_."J1.3.1"] :=
	        DB_UDI.EmptyLine.DownstreamAcu.Stop.Conveyor[_."J1.3.2"];
	        
	    END_REGION
	    
	    REGION J1.3.2
	        //J1.3.2
	        DB_UDI.EmptyLine.DownstreamAcu.Stop.Conveyor[_."J1.3.2"] :=
	        DB_UDI.EmptyLine.DownstreamAcu.Stop.Conveyor[_."J1.4.1"];
	        
	    END_REGION
	    
	    REGION J1.4.1
	        //J1.4.1
	        DB_UDI.EmptyLine.DownstreamAcu.Stop.Conveyor[_."J1.4.1"] :=
	        DB_UDI.EmptyLine.DownstreamAcu.Stop.Conveyor[_."J1.4.2"];
	        
	    END_REGION
	    
	    REGION J1.4.2
	        //J1.4.2
	        DB_UDI.EmptyLine.DownstreamAcu.Stop.Conveyor[_."J1.4.2"] :=
	        DB_UDI.EmptyLine.DownstreamAcu.Stop.Conveyor[_."J1.4.3"];
	        
	    END_REGION
	    
	    REGION J1.4.3
	        //J1.4.3
	        DB_UDI.EmptyLine.DownstreamAcu.Stop.Conveyor[_."J1.4.3"] :=
	        DB_UDI.EmptyLine.DownstreamAcu.Stop.Conveyor[_."J1.4.4"];
	        
	    END_REGION
	    
	    REGION J1.4.4
	        //J1.4.4
	        DB_UDI.EmptyLine.DownstreamAcu.Stop.Conveyor[_."J1.4.4"] :=
	        DB_UDI.EmptyLine.DownstreamAcu.Stop.Conveyor[_."J1.4.5"];
	        
	    END_REGION
	    
	    REGION J1.4.5
	        //J1.4.5
	        DB_UDI.EmptyLine.DownstreamAcu.Stop.Conveyor[_."J1.4.5"] :=
	        DB_UDI.EmptyLine.DownstreamAcu.Stop.Conveyor[_."J1.4.6"];
	        
	    END_REGION
	    
	    REGION J1.4.6
	        //J1.4.6
	        DB_UDI.EmptyLine.DownstreamAcu.Stop.Conveyor[_."J1.4.6"] :=
	        DB_UDI.EmptyLine.DownstreamAcu.Stop.Conveyor[_."J1.4.7"];
	        
	    END_REGION
	    
	    REGION J1.4.7
	        //J1.4.7
	        DB_UDI.EmptyLine.DownstreamAcu.Stop.Conveyor[_."J1.4.7"] :=
	        IDB_EmptyLine."J1.5.1".FilteredSensor OR
	        NOT IDB_EmptyLine."J1.5.1".ReadConveyorStatus.ReadytoRun;
	        
	    END_REGION
	END_REGION
	
	
	REGION J1.5.1
	    //J1.5.1
	    DB_UDI.EmptyLine.DownstreamAcu.Stop.Conveyor[_."J1.5.1"] :=
	    IDB_EmptyLine."J1.5.2".FilteredSensor OR
	    NOT IDB_EmptyLine."J1.5.2".ReadConveyorStatus.ReadytoRun;
	    
	END_REGION
	
	REGION J1.5.2
	    //J1.5.2
	    DB_UDI.EmptyLine.DownstreamAcu.Stop.Conveyor[_."J1.5.2"] :=
	    IDB_EmptyLine."J1.5.3".FilteredSensor OR
	    NOT IDB_EmptyLine."J1.5.3".ReadConveyorStatus.ReadytoRun;
	    
	END_REGION
	
	REGION J1.5.3
	    //J1.5.3
	    DB_UDI.EmptyLine.DownstreamAcu.Stop.Conveyor[_."J1.5.3"] :=
	    IDB_EmptyLine."J1.5.4".FilteredSensor OR
	    NOT IDB_EmptyLine."J1.5.4".ReadConveyorStatus.ReadytoRun;
	    
	END_REGION
	
	REGION J1.5.4
	    //J1.5.4
	    DB_UDI.EmptyLine.DownstreamAcu.Stop.Conveyor[_."J1.5.4"] :=
	    //Straight 
	    (ToteDir.Conveyor[_."J1.6.1"].Straight AND
	    ToteDir.Conveyor[_."J1.6.2"].Straight AND
	    (IDB_EmptyLine."J1.7.1".FilteredSensor OR
	    NOT IDB_EmptyLine."J1.7.1".ReadConveyorStatus.ReadytoRun)) OR
	    //Left
	    (ToteDir.Conveyor[_."J1.6.1"].toLeft AND
	    ToteDir.Conveyor[_."J1.6.2"].toLeft AND
	    (IDB_EmptyLine."J1.2.1".FilteredSensor OR
	    NOT IDB_EmptyLine."K1.1.1".ReadConveyorStatus.ReadytoRun OR
	    NOT IDB_EmptyLine."K1.2.1".ReadConveyorStatus.ReadytoRun)) OR
	    IDB_EmptyLine."J1.6.1".ReadMabsStatus.ReadytoRun OR
	    IDB_EmptyLine."J1.6.2".ReadMabsStatus.ReadytoRun;
	    
	END_REGION
	
	(* REGION J1.6.1 Mabs
	    //Mabs J1.6.1
	    DB_UDI.EmptyLine.DownstreamAcu.Stop.Conveyor[_."J1.6.1"] :=
	    IDB_EmptyLine."J1.6.2".FilteredSensor OR
	    NOT IDB_EmptyLine."J1.6.2".ReadMabsStatus.ReadytoRun;
	    
	END_REGION
	
	REGION J1.6.2 Mabs
	    //Mabs J1.6.2
	    DB_UDI.EmptyLine.DownstreamAcu.Stop.Conveyor[_."J1.6.2"] :=
	    IDB_EmptyLine."J1.7.1".FilteredSensor OR
	    NOT IDB_EmptyLine."J1.7.1".ReadConveyorStatus.ReadytoRun;
	    
	END_REGION *)
	
	REGION J1.7.1 (Go straight )
	    //J1.7.1 (Go straight )
	    DB_UDI.EmptyLine.DownstreamAcu.Stop.Conveyor[_."J1.7.1"] :=
	    IDB_EmptyLine."J1.7.2".FilteredSensor OR
	    NOT IDB_EmptyLine."J1.7.2".ReadConveyorStatus.ReadytoRun;
	    
	END_REGION
	
	REGION J1.7.2
	    //J1.7.2
	    DB_UDI.EmptyLine.DownstreamAcu.Stop.Conveyor[_."J1.7.2"] :=
	    IDB_EmptyLine."J1.8.1".FilteredSensor OR
	    NOT IDB_EmptyLine."J1.8.1".ReadConveyorStatus.ReadytoRun;
	    
	END_REGION
	
	REGION J1.8.1
	    //J1.8.1
	    DB_UDI.EmptyLine.DownstreamAcu.Stop.Conveyor[_."J1.8.1"] :=
	    IDB_EmptyLine."J1.8.2".FilteredSensor OR
	    NOT IDB_EmptyLine."J1.8.2".ReadConveyorStatus.ReadytoRun;
	    
	END_REGION
	
	REGION J1.8.2
	    //J1.8.2
	    DB_UDI.EmptyLine.DownstreamAcu.Stop.Conveyor[_."J1.8.2"] :=
	    IDB_EmptyLine."J1.9.1".FilteredSensor OR
	    NOT IDB_EmptyLine."J1.9.1".ReadConveyorStatus.ReadytoRun;
	    
	END_REGION
	
	REGION J1.9.1
	    //J1.9.1
	    DB_UDI.EmptyLine.DownstreamAcu.Stop.Conveyor[_."J1.9.1"] :=
	    IDB_EmptyLine."J1.10.1".FilteredSensor OR
	    NOT IDB_EmptyLine."J1.10.1".ReadConveyorStatus.ReadytoRun;
	    
	END_REGION
	
	REGION J1.10.1
	    //J1.10.1
	    DB_UDI.EmptyLine.DownstreamAcu.Stop.Conveyor[_."J1.10.1"] :=
	    IDB_EmptyLine."J1.11.7".FilteredSensor OR
	    NOT IDB_EmptyLine."J1.11.1".ReadConveyorStatus.ReadytoRun OR
	    NOT IDB_EmptyLine."J1.11.2".ReadConveyorStatus.ReadytoRun OR
	    NOT IDB_EmptyLine."J1.11.3".ReadConveyorStatus.ReadytoRun OR
	    NOT IDB_EmptyLine."J1.11.4".ReadConveyorStatus.ReadytoRun OR
	    NOT IDB_EmptyLine."J1.11.5".ReadConveyorStatus.ReadytoRun OR
	    NOT IDB_EmptyLine."J1.11.6".ReadConveyorStatus.ReadytoRun OR
	    NOT IDB_EmptyLine."J1.11.7".ReadConveyorStatus.ReadytoRun;
	    
	END_REGION
	
	REGION J1.11.1 TO J1.11.7
	    REGION J1.11.1
	        //J1.11.1
	        DB_UDI.EmptyLine.DownstreamAcu.Stop.Conveyor[_."J1.11.1"] :=
	        DB_UDI.EmptyLine.DownstreamAcu.Stop.Conveyor[_."J1.11.2"];
	        
	    END_REGION
	    
	    REGION J1.11.2
	        //J1.11.2
	        DB_UDI.EmptyLine.DownstreamAcu.Stop.Conveyor[_."J1.11.2"] :=
	        DB_UDI.EmptyLine.DownstreamAcu.Stop.Conveyor[_."J1.11.3"];
	        
	    END_REGION
	    
	    REGION J1.11.3
	        //J1.11.3
	        DB_UDI.EmptyLine.DownstreamAcu.Stop.Conveyor[_."J1.11.3"] :=
	        DB_UDI.EmptyLine.DownstreamAcu.Stop.Conveyor[_."J1.11.4"];
	        
	    END_REGION
	    
	    REGION J1.11.4
	        //J1.11.4
	        DB_UDI.EmptyLine.DownstreamAcu.Stop.Conveyor[_."J1.11.4"] :=
	        DB_UDI.EmptyLine.DownstreamAcu.Stop.Conveyor[_."J1.11.5"];
	        
	    END_REGION
	    
	    REGION J1.11.5
	        //J1.11.5
	        DB_UDI.EmptyLine.DownstreamAcu.Stop.Conveyor[_."J1.11.5"] :=
	        DB_UDI.EmptyLine.DownstreamAcu.Stop.Conveyor[_."J1.11.6"];
	        
	    END_REGION
	    
	    REGION J1.11.6
	        //J1.11.6
	        DB_UDI.EmptyLine.DownstreamAcu.Stop.Conveyor[_."J1.11.6"] :=
	        DB_UDI.EmptyLine.DownstreamAcu.Stop.Conveyor[_."J1.11.7"];
	        
	    END_REGION
	    
	    REGION J1.11.7
	        //J1.11.7
	        DB_UDI.EmptyLine.DownstreamAcu.Stop.Conveyor[_."J1.11.7"] :=
	        IDB_EmptyLine."J1.11.13".FilteredSensor OR
	        NOT IDB_EmptyLine."J1.11.8".ReadConveyorStatus.ReadytoRun OR
	        NOT IDB_EmptyLine."J1.11.9".ReadConveyorStatus.ReadytoRun OR
	        NOT IDB_EmptyLine."J1.11.10".ReadConveyorStatus.ReadytoRun OR
	        NOT IDB_EmptyLine."J1.11.11".ReadConveyorStatus.ReadytoRun OR
	        NOT IDB_EmptyLine."J1.11.12".ReadConveyorStatus.ReadytoRun OR
	        NOT IDB_EmptyLine."J1.11.13".ReadConveyorStatus.ReadytoRun;
	        
	    END_REGION
	END_REGION
	
	
	REGION J1.11.8 TO J1.11.13
	    REGION J1.11.8
	        //J1.11.8
	        DB_UDI.EmptyLine.DownstreamAcu.Stop.Conveyor[_."J1.11.8"] :=
	        DB_UDI.EmptyLine.DownstreamAcu.Stop.Conveyor[_."J1.11.9"];
	        
	    END_REGION
	    
	    REGION J1.11.9
	        //J1.11.9
	        DB_UDI.EmptyLine.DownstreamAcu.Stop.Conveyor[_."J1.11.9"] :=
	        DB_UDI.EmptyLine.DownstreamAcu.Stop.Conveyor[_."J1.11.10"];
	        
	    END_REGION
	    
	    REGION J1.11.10
	        //J1.11.10
	        DB_UDI.EmptyLine.DownstreamAcu.Stop.Conveyor[_."J1.11.10"] :=
	        DB_UDI.EmptyLine.DownstreamAcu.Stop.Conveyor[_."J1.11.11"];
	        
	    END_REGION
	    
	    REGION J1.11.11
	        //J1.11.11
	        DB_UDI.EmptyLine.DownstreamAcu.Stop.Conveyor[_."J1.11.11"] :=
	        DB_UDI.EmptyLine.DownstreamAcu.Stop.Conveyor[_."J1.11.12"];
	        
	    END_REGION
	    
	    REGION J1.11.12
	        //J1.11.12
	        DB_UDI.EmptyLine.DownstreamAcu.Stop.Conveyor[_."J1.11.12"] :=
	        DB_UDI.EmptyLine.DownstreamAcu.Stop.Conveyor[_."J1.11.13"];
	        
	    END_REGION
	    
	    REGION J1.11.13
	        //J1.11.13
	        DB_UDI.EmptyLine.DownstreamAcu.Stop.Conveyor[_."J1.11.13"] :=
	        IDB_EmptyLine."J1.11.13".FilteredSensor;
	        
	    END_REGION
	END_REGION
	
	
	REGION K1.1.1 TO K1.2.1
	    REGION K1.1.1 (Go Left)
	        //K1.1.1  (Go Left)
	        DB_UDI.EmptyLine.DownstreamAcu.Stop.Conveyor[_."K1.1.1"] :=
	        DB_UDI.EmptyLine.DownstreamAcu.Stop.Conveyor[_."K1.2.1"];
	        
	    END_REGION
	    
	    REGION K1.2.1
	        //K1.2.1
	        DB_UDI.EmptyLine.DownstreamAcu.Stop.Conveyor[_."K1.2.1"] :=
	        IDB_EmptyLine."K1.3.1".FilteredSensor OR
	        NOT IDB_EmptyLine."K1.3.1".ReadConveyorStatus.ReadytoRun;
	        
	    END_REGION
	END_REGION
	
	
	REGION K1.3.1
	    //K1.3.1
	    DB_UDI.EmptyLine.DownstreamAcu.Stop.Conveyor[_."K1.3.1"] :=
	    IDB_EmptyLine."K1.4.1".FilteredSensor OR
	    NOT IDB_EmptyLine."K1.4.1".ReadConveyorStatus.ReadytoRun;
	    
	END_REGION
	
	REGION K1.4.1
	    //K1.4.1
	    DB_UDI.EmptyLine.DownstreamAcu.Stop.Conveyor[_."K1.4.1"] :=
	    IDB_EmptyLine."K1.4.10".FilteredSensor OR
	    NOT IDB_EmptyLine."K1.4.2".ReadConveyorStatus.ReadytoRun OR
	    NOT IDB_EmptyLine."K1.4.3".ReadConveyorStatus.ReadytoRun OR
	    NOT IDB_EmptyLine."K1.4.4".ReadConveyorStatus.ReadytoRun OR
	    NOT IDB_EmptyLine."K1.4.5".ReadConveyorStatus.ReadytoRun OR
	    NOT IDB_EmptyLine."K1.4.6".ReadConveyorStatus.ReadytoRun OR
	    NOT IDB_EmptyLine."K1.4.7".ReadConveyorStatus.ReadytoRun OR
	    NOT IDB_EmptyLine."K1.4.8".ReadConveyorStatus.ReadytoRun OR
	    NOT IDB_EmptyLine."K1.4.9".ReadConveyorStatus.ReadytoRun OR
	    NOT IDB_EmptyLine."K1.4.10".ReadConveyorStatus.ReadytoRun;
	    
	END_REGION
	
	REGION K1.4.2 TO K1.4.10
	    REGION K1.4.2
	        //K1.4.2
	        DB_UDI.EmptyLine.DownstreamAcu.Stop.Conveyor[_."K1.4.2"] :=
	        DB_UDI.EmptyLine.DownstreamAcu.Stop.Conveyor[_."K1.4.3"];
	        
	    END_REGION
	    
	    REGION K1.4.3
	        //K1.4.3
	        DB_UDI.EmptyLine.DownstreamAcu.Stop.Conveyor[_."K1.4.3"] :=
	        DB_UDI.EmptyLine.DownstreamAcu.Stop.Conveyor[_."K1.4.4"];
	        
	    END_REGION
	    
	    REGION K1.4.4
	        //K1.4.4
	        DB_UDI.EmptyLine.DownstreamAcu.Stop.Conveyor[_."K1.4.4"] :=
	        DB_UDI.EmptyLine.DownstreamAcu.Stop.Conveyor[_."K1.4.5"];
	        
	    END_REGION
	    
	    REGION K1.4.5
	        //K1.4.5
	        DB_UDI.EmptyLine.DownstreamAcu.Stop.Conveyor[_."K1.4.5"] :=
	        DB_UDI.EmptyLine.DownstreamAcu.Stop.Conveyor[_."K1.4.6"];
	        
	    END_REGION
	    
	    REGION K1.4.6
	        //K1.4.6
	        DB_UDI.EmptyLine.DownstreamAcu.Stop.Conveyor[_."K1.4.6"] :=
	        DB_UDI.EmptyLine.DownstreamAcu.Stop.Conveyor[_."K1.4.7"];
	        
	    END_REGION
	    
	    REGION K1.4.7
	        //K1.4.7
	        DB_UDI.EmptyLine.DownstreamAcu.Stop.Conveyor[_."K1.4.7"] :=
	        DB_UDI.EmptyLine.DownstreamAcu.Stop.Conveyor[_."K1.4.8"];
	        
	    END_REGION
	    
	    REGION K1.4.8
	        //K1.4.8
	        DB_UDI.EmptyLine.DownstreamAcu.Stop.Conveyor[_."K1.4.8"] :=
	        DB_UDI.EmptyLine.DownstreamAcu.Stop.Conveyor[_."K1.4.9"];
	        
	    END_REGION
	    
	    REGION K1.4.9
	        //K1.4.9
	        DB_UDI.EmptyLine.DownstreamAcu.Stop.Conveyor[_."K1.4.9"] :=
	        DB_UDI.EmptyLine.DownstreamAcu.Stop.Conveyor[_."K1.4.10"];
	        
	    END_REGION
	    
	    REGION K1.4.10
	        //K1.4.10
	        DB_UDI.EmptyLine.DownstreamAcu.Stop.Conveyor[_."K1.4.10"] :=
	        IDB_EmptyLine."K1.5.8".FilteredSensor OR
	        NOT IDB_EmptyLine."K1.5.1".ReadConveyorStatus.ReadytoRun OR
	        NOT IDB_EmptyLine."K1.5.2".ReadConveyorStatus.ReadytoRun OR
	        NOT IDB_EmptyLine."K1.5.3".ReadConveyorStatus.ReadytoRun OR
	        NOT IDB_EmptyLine."K1.5.4".ReadConveyorStatus.ReadytoRun OR
	        NOT IDB_EmptyLine."K1.5.5".ReadConveyorStatus.ReadytoRun OR
	        NOT IDB_EmptyLine."K1.5.6".ReadConveyorStatus.ReadytoRun OR
	        NOT IDB_EmptyLine."K1.5.7".ReadConveyorStatus.ReadytoRun OR
	        NOT IDB_EmptyLine."K1.5.8".ReadConveyorStatus.ReadytoRun;
	        
	    END_REGION
	END_REGION
	
	
	REGION K1.5.1 TO K1.5.8
	    REGION K1.5.1
	        //K1.5.1
	        DB_UDI.EmptyLine.DownstreamAcu.Stop.Conveyor[_."K1.5.1"] :=
	        DB_UDI.EmptyLine.DownstreamAcu.Stop.Conveyor[_."K1.5.2"];
	        
	    END_REGION
	    
	    REGION K1.5.2
	        //K1.5.2
	        DB_UDI.EmptyLine.DownstreamAcu.Stop.Conveyor[_."K1.5.2"] :=
	        DB_UDI.EmptyLine.DownstreamAcu.Stop.Conveyor[_."K1.5.3"];
	        
	    END_REGION
	    
	    REGION K1.5.3
	        //K1.5.3
	        DB_UDI.EmptyLine.DownstreamAcu.Stop.Conveyor[_."K1.5.3"] :=
	        DB_UDI.EmptyLine.DownstreamAcu.Stop.Conveyor[_."K1.5.4"];
	        
	    END_REGION
	    
	    REGION K1.5.4
	        //K1.5.4
	        DB_UDI.EmptyLine.DownstreamAcu.Stop.Conveyor[_."K1.5.4"] :=
	        DB_UDI.EmptyLine.DownstreamAcu.Stop.Conveyor[_."K1.5.5"];
	        
	    END_REGION
	    
	    REGION K1.5.5
	        //K1.5.5
	        DB_UDI.EmptyLine.DownstreamAcu.Stop.Conveyor[_."K1.5.5"] :=
	        DB_UDI.EmptyLine.DownstreamAcu.Stop.Conveyor[_."K1.5.6"];
	        
	    END_REGION
	    
	    REGION K1.5.6
	        //K1.5.6
	        DB_UDI.EmptyLine.DownstreamAcu.Stop.Conveyor[_."K1.5.6"] :=
	        DB_UDI.EmptyLine.DownstreamAcu.Stop.Conveyor[_."K1.5.7"];
	        
	    END_REGION
	    
	    REGION K1.5.7
	        //K1.5.7
	        DB_UDI.EmptyLine.DownstreamAcu.Stop.Conveyor[_."K1.5.7"] :=
	        DB_UDI.EmptyLine.DownstreamAcu.Stop.Conveyor[_."K1.5.8"];
	        
	    END_REGION
	    
	    REGION K1.5.8
	        //K1.5.8
	        DB_UDI.EmptyLine.DownstreamAcu.Stop.Conveyor[_."K1.5.8"] :=
	        IDB_EmptyLine."K1.6.1".FilteredSensor OR
	        NOT IDB_EmptyLine."K1.6.1".ReadConveyorStatus.ReadytoRun;
	        
	    END_REGION
	END_REGION
	
	
	REGION K1.6.1
	    //K1.6.1
	    DB_UDI.EmptyLine.DownstreamAcu.Stop.Conveyor[_."K1.6.1"] :=
	    IDB_EmptyLine."K1.6.2".FilteredSensor OR
	    NOT IDB_EmptyLine."K1.6.2".ReadConveyorStatus.ReadytoRun;
	    
	END_REGION
	
	REGION K1.6.2
	    //K1.6.2
	    DB_UDI.EmptyLine.DownstreamAcu.Stop.Conveyor[_."K1.6.2"] :=
	    IDB_EmptyLine."K1.7.1".FilteredSensor OR
	    NOT IDB_EmptyLine."K1.7.1".ReadConveyorStatus.ReadytoRun;
	    
	END_REGION
	
	REGION K1.7.1 TO K1.7.2
	    REGION K1.7.1
	        //K1.7.1
	        DB_UDI.EmptyLine.DownstreamAcu.Stop.Conveyor[_."K1.7.1"] :=
	        DB_UDI.EmptyLine.DownstreamAcu.Stop.Conveyor[_."K1.7.2"];
	        
	    END_REGION
	    
	    REGION K1.7.2
	        //K1.7.2
	        DB_UDI.EmptyLine.DownstreamAcu.Stop.Conveyor[_."K1.7.2"] :=
	        IDB_EmptyLine."K1.8.3".FilteredSensor OR
	        NOT IDB_EmptyLine."K1.8.1".ReadConveyorStatus.ReadytoRun OR
	        NOT IDB_EmptyLine."K1.8.2".ReadConveyorStatus.ReadytoRun OR
	        NOT IDB_EmptyLine."K1.8.3".ReadConveyorStatus.ReadytoRun;
	        
	    END_REGION
	END_REGION
	
	
	REGION K1.8.1 TO K1.8.3
	    REGION K1.8.1
	        //K1.8.1
	        DB_UDI.EmptyLine.DownstreamAcu.Stop.Conveyor[_."K1.8.1"] :=
	        DB_UDI.EmptyLine.DownstreamAcu.Stop.Conveyor[_."K1.8.2"];
	        
	    END_REGION
	    
	    REGION K1.8.2
	        //K1.8.2
	        DB_UDI.EmptyLine.DownstreamAcu.Stop.Conveyor[_."K1.8.2"] :=
	        DB_UDI.EmptyLine.DownstreamAcu.Stop.Conveyor[_."K1.8.3"];
	        
	    END_REGION
	    
	    REGION K1.8.3
	        //K1.8.3
	        DB_UDI.EmptyLine.DownstreamAcu.Stop.Conveyor[_."K1.8.3"] :=
	        IDB_EmptyLine."K1.10.1".FilteredSensor OR
	        NOT IDB_EmptyLine."K1.9.1".ReadConveyorStatus.ReadytoRun OR
	        NOT IDB_EmptyLine."K1.9.2".ReadConveyorStatus.ReadytoRun OR
	        NOT IDB_EmptyLine."K1.9.3".ReadConveyorStatus.ReadytoRun OR
	        NOT IDB_EmptyLine."K1.9.4".ReadConveyorStatus.ReadytoRun OR
	        NOT IDB_EmptyLine."K1.9.5".ReadConveyorStatus.ReadytoRun OR
	        NOT IDB_EmptyLine."K1.9.6".ReadConveyorStatus.ReadytoRun OR
	        NOT IDB_EmptyLine."K1.9.7".ReadConveyorStatus.ReadytoRun OR
	        NOT IDB_EmptyLine."K1.10.1".ReadConveyorStatus.ReadytoRun;
	        
	    END_REGION
	END_REGION
	
	REGION K1.9.1 TO K1.10.1
	    REGION K1.9.1
	        //K1.9.1
	        DB_UDI.EmptyLine.DownstreamAcu.Stop.Conveyor[_."K1.9.1"] :=
	        DB_UDI.EmptyLine.DownstreamAcu.Stop.Conveyor[_."K1.9.2"];
	        
	    END_REGION
	    
	    REGION K1.9.2
	        //K1.9.2
	        DB_UDI.EmptyLine.DownstreamAcu.Stop.Conveyor[_."K1.9.2"] :=
	        DB_UDI.EmptyLine.DownstreamAcu.Stop.Conveyor[_."K1.9.3"];
	        
	    END_REGION
	    
	    REGION K1.9.3
	        //K1.9.3
	        DB_UDI.EmptyLine.DownstreamAcu.Stop.Conveyor[_."K1.9.3"] :=
	        DB_UDI.EmptyLine.DownstreamAcu.Stop.Conveyor[_."K1.9.4"];
	        
	    END_REGION
	    
	    REGION K1.9.4
	        //K1.9.4
	        DB_UDI.EmptyLine.DownstreamAcu.Stop.Conveyor[_."K1.9.4"] :=
	        DB_UDI.EmptyLine.DownstreamAcu.Stop.Conveyor[_."K1.9.5"];
	        
	    END_REGION
	    
	    REGION K1.9.5
	        //K1.9.5
	        DB_UDI.EmptyLine.DownstreamAcu.Stop.Conveyor[_."K1.9.5"] :=
	        DB_UDI.EmptyLine.DownstreamAcu.Stop.Conveyor[_."K1.9.6"];
	        
	    END_REGION
	    
	    REGION K1.9.6
	        //K1.9.6
	        DB_UDI.EmptyLine.DownstreamAcu.Stop.Conveyor[_."K1.9.6"] :=
	        DB_UDI.EmptyLine.DownstreamAcu.Stop.Conveyor[_."K1.9.7"];
	        
	    END_REGION
	    
	    REGION K1.9.7
	        //K1.9.7
	        DB_UDI.EmptyLine.DownstreamAcu.Stop.Conveyor[_."K1.9.7"] :=
	        DB_UDI.EmptyLine.DownstreamAcu.Stop.Conveyor[_."K1.10.1"];
	        
	    END_REGION
	    
	    REGION K1.10.1
	        //K1.10.1
	        DB_UDI.EmptyLine.DownstreamAcu.Stop.Conveyor[_."K1.10.1"] :=
	        IDB_EmptyLine."K1.10.1".FilteredSensor;
	        
	    END_REGION
	END_REGION
	
	
	
END_FUNCTION
END_NAMESPACE

NAMESPACE EmptyLine
FUNCTION FC_Fault : Void
{ S7_Optimized_Access := 'TRUE' ; Published := 'TRUE' }
VERSION : 0.1

BEGIN
	// ==========================================================================================================================================
	// Company        : LogTech, s.r.o.
	// Created by     : Anton Vinoth Soundraraj
	// Block          : FC_Fault
	// Project        : Lékarna DC Chrudim
	// Project number : 23-157
	// ==========================================================================================================================================
	
	// ===== bw143-C1 =====
	REGION J1.1.1
	    //J1.1.1
	    DB_UDI.EmptyLine.Fault.Stop.Conveyor[_."J1.1.1"] :=
	    _."ASiGW-MCC001-bw143-C1: Input"."Error J1.1.1" OR
	    _."ASiGW-MCC001-bw143-C1: ConfigErr".Slave."18B" OR
	    _."ASiGW-MCC001-bw143-C1: PeriErr".Slave."18B" OR
	    _.Global.IDB_HardwareDiag."BW-ASi -10.106.129.143".CommunicationError;
	    
	END_REGION
	
	// ===== bw143-C1 =====
	REGION J1.1.2
	    //J1.1.2
	    DB_UDI.EmptyLine.Fault.Stop.Conveyor[_."J1.1.2"] :=
	    _."ASiGW-MCC001-bw143-C1: Input"."Error J1.1.2" OR
	    _."ASiGW-MCC001-bw143-C1: ConfigErr".Slave."18B" OR
	    _."ASiGW-MCC001-bw143-C1: PeriErr".Slave."18B" OR
	    _.Global.IDB_HardwareDiag."BW-ASi -10.106.129.143".CommunicationError;
	    
	END_REGION
	
	// ===== bw143-C1 =====
	REGION J1.1.3
	    //J1.1.3
	    DB_UDI.EmptyLine.Fault.Stop.Conveyor[_."J1.1.3"] :=
	    _."ASiGW-MCC001-bw143-C1: Input"."Error J1.1.3" OR
	    _."ASiGW-MCC001-bw143-C1: ConfigErr".Slave."19B" OR
	    _."ASiGW-MCC001-bw143-C1: PeriErr".Slave."19B" OR
	    _.Global.IDB_HardwareDiag."BW-ASi -10.106.129.143".CommunicationError;
	    
	END_REGION
	
	// ===== bw143-C1 =====
	REGION J1.1.4
	    //J1.1.4
	    DB_UDI.EmptyLine.Fault.Stop.Conveyor[_."J1.1.4"] :=
	    _."ASiGW-MCC001-bw143-C1: Input"."Error J1.1.4" OR
	    _."ASiGW-MCC001-bw143-C1: ConfigErr".Slave."19B" OR
	    _."ASiGW-MCC001-bw143-C1: PeriErr".Slave."19B" OR
	    _.Global.IDB_HardwareDiag."BW-ASi -10.106.129.143".CommunicationError;
	    
	END_REGION
	
	// ===== bw143-C1 =====
	REGION J1.1.5
	    //J1.1.5
	    DB_UDI.EmptyLine.Fault.Stop.Conveyor[_."J1.1.5"] :=
	    _."ASiGW-MCC001-bw143-C1: Input"."Error J1.1.5" OR
	    _."ASiGW-MCC001-bw143-C1: ConfigErr".Slave."20B" OR
	    _."ASiGW-MCC001-bw143-C1: PeriErr".Slave."20B" OR
	    _.Global.IDB_HardwareDiag."BW-ASi -10.106.129.143".CommunicationError;
	    
	END_REGION
	
	// ===== bw143-C1 =====
	REGION J1.1.6
	    //J1.1.6
	    DB_UDI.EmptyLine.Fault.Stop.Conveyor[_."J1.1.6"] :=
	    _."ASiGW-MCC001-bw143-C1: Input"."Error J1.1.6" OR
	    _."ASiGW-MCC001-bw143-C1: ConfigErr".Slave."20B" OR
	    _."ASiGW-MCC001-bw143-C1: PeriErr".Slave."20B" OR
	    _.Global.IDB_HardwareDiag."BW-ASi -10.106.129.143".CommunicationError;
	    
	END_REGION
	
	// ===== bw143-C1 =====
	REGION J1.1.7
	    //J1.1.7
	    DB_UDI.EmptyLine.Fault.Stop.Conveyor[_."J1.1.7"] :=
	    _."ASiGW-MCC001-bw143-C1: Input"."Error J1.1.7" OR
	    _."ASiGW-MCC001-bw143-C1: ConfigErr".Slave."21B" OR
	    _."ASiGW-MCC001-bw143-C1: PeriErr".Slave."21B" OR
	    _.Global.IDB_HardwareDiag."BW-ASi -10.106.129.143".CommunicationError;
	    
	END_REGION
	
	// ===== bw143-C1 =====
	REGION J1.1.8
	    //J1.1.8
	    DB_UDI.EmptyLine.Fault.Stop.Conveyor[_."J1.1.8"] :=
	    _."ASiGW-MCC001-bw143-C1: Input"."Error J1.1.8" OR
	    _."ASiGW-MCC001-bw143-C1: ConfigErr".Slave."21B" OR
	    _."ASiGW-MCC001-bw143-C1: PeriErr".Slave."21B" OR
	    _.Global.IDB_HardwareDiag."BW-ASi -10.106.129.143".CommunicationError;
	    
	END_REGION
	
	// ===== bw143-C1 =====
	REGION J1.1.9
	    //J1.1.9
	    DB_UDI.EmptyLine.Fault.Stop.Conveyor[_."J1.1.9"] :=
	    _."ASiGW-MCC001-bw143-C1: Input"."Error J1.1.9" OR
	    _."ASiGW-MCC001-bw143-C1: ConfigErr".Slave."22B" OR
	    _."ASiGW-MCC001-bw143-C1: PeriErr".Slave."22B" OR
	    _.Global.IDB_HardwareDiag."BW-ASi -10.106.129.143".CommunicationError;
	    
	END_REGION
	
	// ===== bw143-C1 =====
	REGION J1.1.10
	    //J1.1.10
	    DB_UDI.EmptyLine.Fault.Stop.Conveyor[_."J1.1.10"] :=
	    _."ASiGW-MCC001-bw143-C1: Input"."Error J1.1.10" OR
	    _."ASiGW-MCC001-bw143-C1: ConfigErr".Slave."22B" OR
	    _."ASiGW-MCC001-bw143-C1: PeriErr".Slave."22B" OR
	    _.Global.IDB_HardwareDiag."BW-ASi -10.106.129.143".CommunicationError;
	    
	END_REGION
	
	// ===== bw143-C1 =====
	REGION J1.1.11
	    //J1.1.11
	    DB_UDI.EmptyLine.Fault.Stop.Conveyor[_."J1.1.11"] :=
	    _."ASiGW-MCC001-bw143-C1: Input"."Error J1.1.11" OR
	    _."ASiGW-MCC001-bw143-C1: ConfigErr".Slave."23B" OR
	    _."ASiGW-MCC001-bw143-C1: PeriErr".Slave."23B" OR
	    _.Global.IDB_HardwareDiag."BW-ASi -10.106.129.143".CommunicationError;
	    
	END_REGION
	
	// ===== bw143-C1 =====
	REGION J1.1.12
	    //J1.1.12
	    DB_UDI.EmptyLine.Fault.Stop.Conveyor[_."J1.1.12"] :=
	    _."ASiGW-MCC001-bw143-C1: Input"."Error J1.1.12" OR
	    _."ASiGW-MCC001-bw143-C1: ConfigErr".Slave."23B" OR
	    _."ASiGW-MCC001-bw143-C1: PeriErr".Slave."23B" OR
	    _.Global.IDB_HardwareDiag."BW-ASi -10.106.129.143".CommunicationError;
	    
	END_REGION
	
	// ===== bw143-C1 =====
	REGION J1.1.13
	    //J1.1.13
	    DB_UDI.EmptyLine.Fault.Stop.Conveyor[_."J1.1.13"] :=
	    _."ASiGW-MCC001-bw143-C1: Input"."Error J1.1.13" OR
	    _."ASiGW-MCC001-bw143-C1: ConfigErr".Slave."24B" OR
	    _."ASiGW-MCC001-bw143-C1: PeriErr".Slave."24B" OR
	    _.Global.IDB_HardwareDiag."BW-ASi -10.106.129.143".CommunicationError;
	    
	END_REGION
	
	// ===== bw143-C1 =====
	REGION J1.1.14
	    //J1.1.14
	    DB_UDI.EmptyLine.Fault.Stop.Conveyor[_."J1.1.14"] :=
	    _."ASiGW-MCC001-bw143-C1: Input"."Error J1.1.14" OR
	    _."ASiGW-MCC001-bw143-C1: ConfigErr".Slave."24B" OR
	    _."ASiGW-MCC001-bw143-C1: PeriErr".Slave."24B" OR
	    _.Global.IDB_HardwareDiag."BW-ASi -10.106.129.143".CommunicationError;
	    
	END_REGION
	
	// ===== bw143-C1 =====
	REGION J1.1.15
	    //J1.1.15
	    DB_UDI.EmptyLine.Fault.Stop.Conveyor[_."J1.1.15"] :=
	    _."ASiGW-MCC001-bw143-C1: Input"."Error J1.1.15" OR
	    _."ASiGW-MCC001-bw143-C1: ConfigErr".Slave."25B" OR
	    _."ASiGW-MCC001-bw143-C1: PeriErr".Slave."25B" OR
	    _.Global.IDB_HardwareDiag."BW-ASi -10.106.129.143".CommunicationError;
	    
	END_REGION
	
	// ===== bw143-C1 =====
	REGION J1.2.1
	    //J1.2.1
	    DB_UDI.EmptyLine.Fault.Stop.Conveyor[_."J1.2.1"] :=
	    _."ASiGW-MCC001-bw143-C1: Input"."Error J1.2.1" OR
	    _."ASiGW-MCC001-bw143-C1: ConfigErr".Slave."25B" OR
	    _."ASiGW-MCC001-bw143-C1: PeriErr".Slave."25B" OR
	    _.Global.IDB_HardwareDiag."BW-ASi -10.106.129.143".CommunicationError;
	    
	END_REGION
	
	// ===== bw143-C1 =====
	REGION J1.2.2
	    //J1.2.2
	    DB_UDI.EmptyLine.Fault.Stop.Conveyor[_."J1.2.2"] :=
	    _."ASiGW-MCC001-bw143-C1: Input"."Error J1.2.2" OR
	    _."ASiGW-MCC001-bw143-C1: ConfigErr".Slave."26B" OR
	    _."ASiGW-MCC001-bw143-C1: PeriErr".Slave."26B" OR
	    _.Global.IDB_HardwareDiag."BW-ASi -10.106.129.143".CommunicationError;
	    
	END_REGION
	
	// ===== bw143-C1 =====
	REGION J1.2.3
	    //J1.2.3 Staright for Merger1
	    DB_UDI.EmptyLine.Fault.Stop.Conveyor[_."J1.2.3"] :=
	    _."ASiGW-MCC001-bw143-C1: Input"."Error J1.2.3" OR
	    _."ASiGW-MCC001-bw143-C1: ConfigErr".Slave."26B" OR
	    _."ASiGW-MCC001-bw143-C1: PeriErr".Slave."26B" OR
	    _.Global.IDB_HardwareDiag."BW-ASi -10.106.129.143".CommunicationError;
	    
	END_REGION
	
	
	// ===== bw200-C2 =====
	REGION J2.1.1
	    //J2.1.1
	    DB_UDI.EmptyLine.Fault.Stop.Conveyor[_."J2.1.1"] :=
	    _."ASiGW-MCC001-bw200-C2: Input"."Error J2.1.1" OR
	    _."ASiGW-MCC001-bw200-C2: ConfigErr".Slave."16A" OR
	    _."ASiGW-MCC001-bw200-C2: PeriErr".Slave."16A" OR
	    _.Global.IDB_HardwareDiag."BW-ASi -10.106.129.200".CommunicationError;
	    
	END_REGION
	
